C05479=1196.895,313.381,-70.607,-176.497,7.558,148.421
C05480=1196.891,313.629,-70.637,-176.494,7.561,148.421
C05481=1196.886,313.877,-70.668,-176.492,7.564,148.421
C05482=1196.882,314.126,-70.699,-176.490,7.566,148.421
C05483=1196.878,314.401,-70.733,-176.487,7.570,148.421
C05484=1196.873,314.678,-70.767,-176.484,7.573,148.421
C05485=1196.868,314.954,-70.801,-176.481,7.576,148.421
C05486=1196.864,315.230,-70.836,-176.479,7.579,148.421
C05487=1196.860,315.479,-70.867,-176.476,7.583,148.421
C05488=1196.855,315.727,-70.898,-176.474,7.585,148.421
C05489=1196.851,315.974,-70.928,-176.472,7.588,148.421
C05490=1196.847,316.223,-70.959,-176.469,7.591,148.422
C05491=1196.843,316.471,-70.990,-176.467,7.594,148.422
C05492=1196.838,316.719,-71.020,-176.465,7.596,148.422
C05493=1196.834,316.968,-71.051,-176.462,7.599,148.422
C05494=1196.830,317.215,-71.082,-176.460,7.603,148.422
C05495=1196.825,317.463,-71.112,-176.457,7.606,148.422
C05496=1196.822,317.711,-71.144,-176.455,7.608,148.422
C05497=1196.817,317.959,-71.175,-176.453,7.611,148.422
C05498=1196.812,318.207,-71.206,-176.450,7.614,148.422
C05499=1196.809,318.455,-71.236,-176.448,7.617,148.422
C05500=1196.805,318.703,-71.267,-176.445,7.620,148.422
C05501=1196.800,318.951,-71.298,-176.443,7.623,148.422
C05502=1196.796,319.199,-71.330,-176.440,7.626,148.422
C05503=1196.792,319.447,-71.360,-176.438,7.628,148.422
C05504=1196.788,319.696,-71.392,-176.436,7.631,148.422
C05505=1196.783,319.944,-71.422,-176.433,7.634,148.422
C05506=1196.779,320.191,-71.454,-176.431,7.638,148.422
C05507=1196.775,320.440,-71.484,-176.429,7.640,148.422
C05508=1196.771,320.688,-71.515,-176.426,7.643,148.422
C05509=1196.767,320.936,-71.547,-176.424,7.646,148.423
C05510=1196.763,321.184,-71.578,-176.421,7.649,148.423
C05511=1196.758,321.432,-71.609,-176.419,7.652,148.423
C05512=1196.754,321.680,-71.640,-176.417,7.655,148.423
C05513=1196.750,321.928,-71.671,-176.414,7.658,148.423
C05514=1196.746,322.176,-71.702,-176.412,7.661,148.423
C05515=1196.741,322.424,-71.734,-176.410,7.663,148.423
C05516=1196.737,322.672,-71.765,-176.407,7.667,148.423
C05517=1196.733,322.920,-71.796,-176.405,7.670,148.423
C05518=1196.729,323.168,-71.827,-176.402,7.673,148.423
C05519=1196.725,323.416,-71.859,-176.400,7.675,148.423
C05520=1196.720,323.664,-71.890,-176.398,7.678,148.423
C05521=1196.716,323.912,-71.921,-176.395,7.682,148.423
C05522=1196.712,324.160,-71.952,-176.393,7.685,148.423
C05523=1196.708,324.408,-71.983,-176.391,7.687,148.424
C05524=1196.703,324.656,-72.015,-176.388,7.690,148.424
C05525=1196.700,324.904,-72.047,-176.386,7.694,148.424
C05526=1196.695,325.152,-72.078,-176.383,7.697,148.424
C05527=1196.691,325.400,-72.109,-176.381,7.699,148.424
C05528=1196.687,325.648,-72.140,-176.379,7.702,148.424
C05529=1196.683,325.896,-72.172,-176.376,7.705,148.424
C05530=1196.678,326.144,-72.203,-176.374,7.708,148.424
C05531=1196.675,326.392,-72.235,-176.372,7.711,148.424
C05532=1196.669,326.640,-72.266,-176.370,7.714,148.424
C05533=1196.666,326.888,-72.298,-176.367,7.717,148.424
C05534=1196.662,327.136,-72.330,-176.365,7.720,148.425
C05535=1196.657,327.384,-72.360,-176.362,7.723,148.425
C05536=1196.654,327.632,-72.392,-176.360,7.726,148.425
C05537=1196.649,327.879,-72.424,-176.358,7.729,148.425
C05538=1196.645,328.128,-72.455,-176.356,7.732,148.425
C05539=1196.641,328.375,-72.486,-176.353,7.735,148.425
C05540=1196.637,328.624,-72.519,-176.351,7.738,148.425
C05541=1196.632,328.871,-72.550,-176.349,7.741,148.425
C05542=1196.628,329.120,-72.581,-176.346,7.744,148.425
C05543=1196.625,329.368,-72.613,-176.344,7.747,148.425
C05544=1196.620,329.615,-72.645,-176.342,7.750,148.425
C05545=1196.616,329.863,-72.677,-176.340,7.753,148.426
C05546=1196.611,330.111,-72.708,-176.337,7.756,148.426
C05547=1196.607,330.359,-72.740,-176.335,7.759,148.426
C05548=1196.603,330.607,-72.771,-176.333,7.761,148.426
C05549=1196.599,330.855,-72.804,-176.330,7.765,148.426
C05550=1196.595,331.103,-72.836,-176.328,7.768,148.426
C05551=1196.590,331.351,-72.866,-176.325,7.771,148.426
C05552=1196.587,331.599,-72.898,-176.324,7.774,148.426
C05553=1196.582,331.847,-72.930,-176.321,7.777,148.426
C05554=1196.578,332.095,-72.962,-176.319,7.780,148.427
C05555=1196.574,332.343,-72.994,-176.317,7.783,148.427
C05556=1196.570,332.590,-73.025,-176.314,7.786,148.427
C05557=1196.565,332.838,-73.058,-176.312,7.789,148.427
C05558=1196.562,333.086,-73.090,-176.310,7.792,148.427
C05559=1196.557,333.334,-73.121,-176.307,7.795,148.427
C05560=1196.553,333.582,-73.154,-176.305,7.799,148.427
C05561=1196.549,333.831,-73.185,-176.303,7.801,148.428
C05562=1196.545,334.078,-73.216,-176.301,7.804,148.428
C05563=1196.540,334.327,-73.249,-176.298,7.807,148.428
C05564=1196.537,334.575,-73.280,-176.296,7.811,148.428
C05565=1196.531,334.822,-73.313,-176.294,7.813,148.428
C05566=1196.528,335.070,-73.345,-176.292,7.816,148.428
C05567=1196.524,335.318,-73.377,-176.290,7.820,148.428
C05568=1196.519,335.565,-73.409,-176.287,7.823,148.428
C05569=1196.516,335.813,-73.441,-176.285,7.826,148.429
C05570=1196.512,336.061,-73.473,-176.283,7.828,148.429
C05571=1196.507,336.309,-73.505,-176.280,7.831,148.429
C05572=1196.503,336.557,-73.537,-176.278,7.835,148.429
C05573=1196.499,336.805,-73.569,-176.276,7.838,148.429
C05574=1196.495,337.053,-73.601,-176.274,7.841,148.429
C05575=1196.490,337.301,-73.633,-176.272,7.844,148.429
C05576=1196.486,337.549,-73.665,-176.269,7.847,148.430
C05577=1196.482,337.797,-73.698,-176.267,7.850,148.430
C05578=1196.478,338.045,-73.730,-176.265,7.853,148.430
C05579=1196.474,338.292,-73.761,-176.263,7.856,148.430
C05580=1196.470,338.541,-73.794,-176.260,7.859,148.430
C05581=1196.466,338.789,-73.826,-176.258,7.862,148.431
C05582=1196.462,339.036,-73.859,-176.256,7.866,148.431
C05583=1196.458,339.284,-73.890,-176.254,7.868,148.431
C05584=1196.453,339.532,-73.923,-176.252,7.871,148.431
C05585=1196.449,339.780,-73.955,-176.249,7.875,148.431
C05586=1196.445,340.028,-73.988,-176.247,7.878,148.431
C05587=1196.440,340.306,-74.023,-176.245,7.881,148.432
C05588=1196.435,340.585,-74.060,-176.243,7.885,148.432
C05589=1196.431,340.863,-74.096,-176.240,7.888,148.432
C05590=1196.426,341.142,-74.133,-176.237,7.892,148.432
C05591=1196.421,341.390,-74.165,-176.236,7.894,148.432
C05592=1196.418,341.637,-74.198,-176.233,7.898,148.432
C05593=1196.414,341.885,-74.230,-176.231,7.901,148.433
C05594=1196.410,342.133,-74.262,-176.229,7.904,148.433
C05595=1196.406,342.381,-74.295,-176.227,7.907,148.433
C05596=1196.401,342.629,-74.327,-176.225,7.910,148.433
C05597=1196.397,342.877,-74.359,-176.223,7.914,148.434
C05598=1196.393,343.125,-74.392,-176.221,7.917,148.434
C05599=1196.388,343.373,-74.424,-176.218,7.919,148.434
C05600=1196.385,343.620,-74.457,-176.216,7.922,148.434
C05601=1196.381,343.869,-74.489,-176.214,7.926,148.434
C05602=1196.376,344.116,-74.522,-176.212,7.929,148.434
C05603=1196.372,344.364,-74.554,-176.210,7.932,148.435
C05604=1196.368,344.611,-74.587,-176.208,7.935,148.435
C05605=1196.364,344.860,-74.620,-176.206,7.938,148.435
C05606=1196.360,345.107,-74.652,-176.203,7.942,148.435
C05607=1196.356,345.356,-74.685,-176.201,7.945,148.435
C05608=1196.352,345.603,-74.718,-176.199,7.947,148.436
C05609=1196.347,345.851,-74.749,-176.197,7.951,148.436
C05610=1196.343,346.098,-74.783,-176.195,7.954,148.436
C05611=1196.339,346.346,-74.816,-176.193,7.957,148.436
C05612=1196.335,346.594,-74.848,-176.191,7.960,148.436
C05613=1196.331,346.842,-74.881,-176.189,7.963,148.437
C05614=1196.327,347.090,-74.913,-176.187,7.967,148.437
C05615=1196.323,347.338,-74.946,-176.184,7.970,148.437
C05616=1196.318,347.586,-74.979,-176.183,7.972,148.437
C05617=1196.315,347.834,-75.011,-176.180,7.976,148.438
C05618=1196.311,348.081,-75.044,-176.178,7.979,148.438
C05619=1196.306,348.328,-75.077,-176.176,7.983,148.438
C05620=1196.301,348.577,-75.110,-176.175,7.985,148.438
C05621=1196.297,348.825,-75.143,-176.172,7.989,148.439
C05622=1196.294,349.072,-75.175,-176.170,7.992,148.439
C05623=1196.289,349.320,-75.208,-176.168,7.995,148.439
C05624=1196.285,349.568,-75.241,-176.166,7.999,148.439
C05625=1196.281,349.816,-75.274,-176.164,8.001,148.439
C05626=1196.277,350.064,-75.307,-176.162,8.004,148.440
C05627=1196.273,350.311,-75.340,-176.160,8.008,148.440
C05628=1196.268,350.560,-75.373,-176.158,8.011,148.440
C05629=1196.265,350.807,-75.405,-176.156,8.014,148.440
C05630=1196.261,351.055,-75.439,-176.154,8.017,148.441
C05631=1196.257,351.302,-75.472,-176.152,8.020,148.441
C05632=1196.253,351.550,-75.505,-176.150,8.024,148.441
C05633=1196.248,351.799,-75.537,-176.148,8.027,148.442
C05634=1196.244,352.046,-75.571,-176.146,8.030,148.442
C05635=1196.240,352.294,-75.604,-176.144,8.033,148.442
C05636=1196.236,352.542,-75.637,-176.142,8.037,148.442
C05637=1196.232,352.789,-75.670,-176.140,8.039,148.443
C05638=1196.227,353.037,-75.703,-176.138,8.043,148.443
C05639=1196.224,353.285,-75.736,-176.136,8.046,148.443
C05640=1196.220,353.532,-75.769,-176.134,8.049,148.443
C05641=1196.216,353.780,-75.802,-176.132,8.052,148.444
C05642=1196.212,354.028,-75.835,-176.130,8.056,148.444
C05643=1196.208,354.276,-75.868,-176.128,8.059,148.444
C05644=1196.203,354.523,-75.901,-176.126,8.062,148.444
C05645=1196.199,354.771,-75.935,-176.125,8.065,148.445
C05646=1196.195,355.019,-75.968,-176.122,8.068,148.445
C05647=1196.191,355.266,-76.001,-176.120,8.072,148.445
C05648=1196.187,355.514,-76.034,-176.118,8.075,148.446
C05649=1196.183,355.762,-76.067,-176.117,8.078,148.446
C05650=1196.179,356.010,-76.100,-176.114,8.081,148.446
C05651=1196.174,356.257,-76.134,-176.113,8.085,148.446
C05652=1196.171,356.506,-76.167,-176.110,8.088,148.447
C05653=1196.167,356.754,-76.200,-176.109,8.091,148.447
C05654=1196.163,357.001,-76.233,-176.107,8.094,148.447
C05655=1196.158,357.249,-76.267,-176.105,8.098,148.447
C05656=1196.154,357.497,-76.300,-176.103,8.101,148.448
C05657=1196.149,357.745,-76.333,-176.101,8.104,148.448
C05658=1196.146,357.992,-76.367,-176.099,8.107,148.449
C05659=1196.141,358.240,-76.400,-176.097,8.111,148.449
C05660=1196.137,358.487,-76.434,-176.095,8.114,148.449
C05661=1196.133,358.735,-76.467,-176.094,8.117,148.449
C05662=1196.130,358.984,-76.500,-176.092,8.120,148.450
C05663=1196.126,359.231,-76.534,-176.090,8.124,148.450
C05664=1196.122,359.478,-76.567,-176.088,8.127,148.450
C05665=1196.118,359.726,-76.600,-176.086,8.130,148.451
C05666=1196.113,359.974,-76.634,-176.084,8.134,148.451
C05667=1196.109,360.221,-76.668,-176.082,8.137,148.451
C05668=1196.105,360.469,-76.701,-176.081,8.140,148.452
C05669=1196.101,360.717,-76.735,-176.079,8.143,148.452
C05670=1196.097,360.965,-76.768,-176.077,8.147,148.452
C05671=1196.093,361.212,-76.802,-176.076,8.149,148.453
C05672=1196.088,361.460,-76.836,-176.074,8.153,148.453
C05673=1196.084,361.708,-76.869,-176.072,8.156,148.453
C05674=1196.080,361.955,-76.903,-176.070,8.159,148.454
C05675=1196.077,362.204,-76.936,-176.068,8.163,148.454
C05676=1196.073,362.451,-76.969,-176.067,8.166,148.454
C05677=1196.068,362.699,-77.004,-176.065,8.169,148.455
C05678=1196.064,362.946,-77.037,-176.063,8.172,148.455
C05679=1196.060,363.194,-77.070,-176.061,8.176,148.456
C05680=1196.057,363.442,-77.104,-176.060,8.179,148.456
C05681=1196.052,363.690,-77.137,-176.058,8.182,148.456
C05682=1196.048,363.937,-77.172,-176.057,8.185,148.457
C05683=1196.044,364.185,-77.205,-176.055,8.189,148.457
C05684=1196.040,364.432,-77.239,-176.053,8.192,148.457
C05685=1196.036,364.680,-77.272,-176.051,8.195,148.458
C05686=1196.032,364.928,-77.307,-176.050,8.198,148.458
C05687=1196.028,365.176,-77.340,-176.048,8.201,148.458
C05688=1196.024,365.423,-77.374,-176.047,8.205,148.459
C05689=1196.020,365.671,-77.408,-176.045,8.208,148.459
C05690=1196.016,365.918,-77.442,-176.044,8.211,148.460
C05691=1196.011,366.200,-77.480,-176.041,8.215,148.460
C05692=1196.006,366.480,-77.518,-176.040,8.218,148.460
C05693=1196.002,366.762,-77.557,-176.038,8.222,148.461
C05694=1195.998,367.042,-77.595,-176.036,8.226,148.461
C05695=1195.993,367.290,-77.629,-176.034,8.229,148.462
C05696=1195.989,367.537,-77.663,-176.033,8.232,148.462
C05697=1195.985,367.786,-77.697,-176.031,8.235,148.462
C05698=1195.981,368.033,-77.731,-176.030,8.238,148.463
C05699=1195.977,368.280,-77.764,-176.028,8.242,148.463
C05700=1195.972,368.528,-77.798,-176.027,8.245,148.464
C05701=1195.969,368.776,-77.832,-176.025,8.248,148.464
C05702=1195.965,369.023,-77.866,-176.024,8.251,148.465
C05703=1195.960,369.271,-77.900,-176.022,8.255,148.465
C05704=1195.957,369.519,-77.934,-176.021,8.258,148.465
C05705=1195.952,369.767,-77.968,-176.019,8.261,148.466
C05706=1195.948,370.014,-78.002,-176.018,8.264,148.466
C05707=1195.944,370.261,-78.036,-176.016,8.268,148.467
C05708=1195.941,370.509,-78.071,-176.015,8.271,148.467
C05709=1195.936,370.757,-78.104,-176.014,8.274,148.468
C05710=1195.932,371.004,-78.138,-176.012,8.277,148.468
C05711=1195.929,371.252,-78.172,-176.011,8.281,148.468
C05712=1195.924,371.500,-78.207,-176.009,8.284,148.469
C05713=1195.920,371.747,-78.240,-176.008,8.286,148.469
C05714=1195.916,371.995,-78.275,-176.006,8.290,148.470
C05715=1195.912,372.243,-78.309,-176.006,8.293,148.470
C05716=1195.908,372.490,-78.343,-176.004,8.297,148.471
C05717=1195.904,372.738,-78.377,-176.002,8.300,148.471
C05718=1195.899,372.986,-78.411,-176.001,8.302,148.471
C05719=1195.896,373.233,-78.445,-175.999,8.306,148.472
C05720=1195.892,373.481,-78.480,-175.999,8.309,148.472
C05721=1195.888,373.728,-78.514,-175.997,8.312,148.473
C05722=1195.884,373.976,-78.549,-175.996,8.316,148.473
C05723=1195.880,374.224,-78.582,-175.994,8.318,148.474
C05724=1195.875,374.471,-78.616,-175.994,8.322,148.474
C05725=1195.872,374.719,-78.651,-175.992,8.325,148.475
C05726=1195.867,374.967,-78.685,-175.991,8.328,148.475
C05727=1195.864,375.214,-78.719,-175.990,8.331,148.476
C05728=1195.860,375.462,-78.754,-175.989,8.334,148.476
C05729=1195.856,375.709,-78.788,-175.987,8.337,148.477
C05730=1195.852,375.957,-78.822,-175.986,8.341,148.477
C05731=1195.847,376.205,-78.857,-175.985,8.343,148.478
C05732=1195.843,376.452,-78.891,-175.983,8.347,148.478
C05733=1195.839,376.700,-78.926,-175.982,8.350,148.479
C05734=1195.835,376.948,-78.959,-175.981,8.353,148.479
C05735=1195.831,377.196,-78.994,-175.980,8.356,148.480
C05736=1195.827,377.443,-79.027,-175.979,8.359,148.480
C05737=1195.823,377.690,-79.062,-175.978,8.363,148.481
C05738=1195.819,377.938,-79.097,-175.976,8.366,148.481
C05739=1195.815,378.185,-79.131,-175.976,8.369,148.482
C05740=1195.811,378.434,-79.165,-175.974,8.371,148.482
C05741=1195.807,378.681,-79.200,-175.974,8.375,148.482
C05742=1195.803,378.927,-79.234,-175.972,8.377,148.483
C05743=1195.799,379.176,-79.269,-175.971,8.381,148.484
C05744=1195.795,379.423,-79.304,-175.970,8.384,148.484
C05745=1195.791,379.671,-79.338,-175.969,8.387,148.485
C05746=1195.787,379.918,-79.372,-175.968,8.390,148.485
C05747=1195.783,380.166,-79.407,-175.967,8.393,148.485
C05748=1195.779,380.413,-79.441,-175.966,8.396,148.486
C05749=1195.775,380.662,-79.476,-175.965,8.399,148.486
C05750=1195.770,380.909,-79.510,-175.964,8.402,148.487
C05751=1195.767,381.156,-79.544,-175.963,8.405,148.487
C05752=1195.763,381.404,-79.579,-175.962,8.408,148.488
C05753=1195.758,381.652,-79.614,-175.961,8.411,148.489
C05754=1195.755,381.899,-79.649,-175.960,8.414,148.489
C05755=1195.750,382.146,-79.683,-175.959,8.417,148.490
C05756=1195.747,382.394,-79.718,-175.959,8.420,148.490
C05757=1195.742,382.642,-79.752,-175.957,8.423,148.491
C05758=1195.739,382.890,-79.787,-175.957,8.426,148.491
C05759=1195.734,383.137,-79.821,-175.956,8.429,148.492
C05760=1195.730,383.384,-79.857,-175.955,8.432,148.492
C05761=1195.727,383.632,-79.891,-175.954,8.435,148.493
C05762=1195.723,383.880,-79.925,-175.953,8.438,148.493
C05763=1195.718,384.127,-79.960,-175.952,8.441,148.494
C05764=1195.714,384.375,-79.995,-175.951,8.444,148.494
C05765=1195.711,384.622,-80.029,-175.950,8.447,148.495
C05766=1195.707,384.870,-80.064,-175.949,8.450,148.495
C05767=1195.702,385.117,-80.099,-175.949,8.453,148.496
C05768=1195.698,385.365,-80.133,-175.947,8.456,148.496
C05769=1195.694,385.612,-80.169,-175.947,8.458,148.497
C05770=1195.691,385.860,-80.203,-175.946,8.461,148.498
C05771=1195.686,386.107,-80.237,-175.946,8.465,148.498
C05772=1195.682,386.355,-80.273,-175.945,8.468,148.499
C05773=1195.678,386.602,-80.307,-175.944,8.471,148.499
C05774=1195.674,386.850,-80.342,-175.943,8.473,148.500
C05775=1195.670,387.098,-80.376,-175.943,8.476,148.500
C05776=1195.666,387.345,-80.412,-175.942,8.479,148.501
C05777=1195.662,387.593,-80.446,-175.941,8.482,148.501
C05778=1195.658,387.841,-80.481,-175.941,8.484,148.502
C05779=1195.654,388.088,-80.516,-175.940,8.487,148.503
C05780=1195.650,388.335,-80.550,-175.939,8.491,148.503
C05781=1195.646,388.583,-80.585,-175.938,8.494,148.504
C05782=1195.642,388.830,-80.620,-175.938,8.496,148.504
C05783=1195.638,389.078,-80.655,-175.937,8.499,148.505
C05784=1195.634,389.325,-80.690,-175.936,8.502,148.505
C05785=1195.630,389.573,-80.725,-175.936,8.504,148.506
C05786=1195.626,389.820,-80.759,-175.935,8.507,148.506
C05787=1195.622,390.068,-80.795,-175.935,8.509,148.507
C05788=1195.618,390.316,-80.829,-175.934,8.513,148.507
C05789=1195.614,390.563,-80.865,-175.933,8.516,148.508
C05790=1195.610,390.811,-80.899,-175.933,8.518,148.509
C05791=1195.606,391.058,-80.934,-175.932,8.521,148.509
C05792=1195.602,391.306,-80.969,-175.932,8.523,148.510
C05793=1195.597,391.553,-81.004,-175.931,8.526,148.510
C05794=1195.594,391.800,-81.039,-175.931,8.529,148.511
C05795=1195.589,392.084,-81.078,-175.930,8.532,148.511
C05796=1195.585,392.367,-81.119,-175.930,8.535,148.512
C05797=1195.580,392.650,-81.158,-175.929,8.538,148.513
C05798=1195.576,392.933,-81.199,-175.928,8.541,148.513
C05799=1195.571,393.181,-81.234,-175.928,8.544,148.514
C05800=1195.568,393.428,-81.269,-175.927,8.547,148.514
C05801=1195.564,393.676,-81.303,-175.927,8.549,148.515
C05802=1195.560,393.923,-81.339,-175.926,8.552,148.516
C05803=1195.556,394.171,-81.373,-175.926,8.554,148.516
C05804=1195.552,394.418,-81.409,-175.925,8.557,148.517
C05805=1195.548,394.666,-81.443,-175.925,8.560,148.517
C05806=1195.544,394.913,-81.479,-175.924,8.563,148.518
C05807=1195.540,395.161,-81.513,-175.924,8.565,148.518
C05808=1195.536,395.408,-81.549,-175.924,8.567,148.519
C05809=1195.531,395.656,-81.583,-175.923,8.570,148.519
C05810=1195.528,395.903,-81.619,-175.923,8.573,148.520
C05811=1195.524,396.151,-81.655,-175.923,8.575,148.521
C05812=1195.519,396.398,-81.689,-175.922,8.578,148.521
C05813=1195.516,396.646,-81.725,-175.922,8.581,148.522
C05814=1195.512,396.894,-81.759,-175.922,8.583,148.522
C05815=1195.508,397.141,-81.795,-175.921,8.586,148.523
C05816=1195.504,397.389,-81.829,-175.921,8.588,148.523
C05817=1195.499,397.636,-81.865,-175.920,8.591,148.524
C05818=1195.496,397.883,-81.900,-175.920,8.594,148.525
C05819=1195.492,398.131,-81.935,-175.919,8.596,148.525
C05820=1195.487,398.378,-81.970,-175.919,8.598,148.526
C05821=1195.483,398.626,-82.005,-175.919,8.600,148.526
C05822=1195.480,398.874,-82.041,-175.918,8.604,148.527
C05823=1195.476,399.120,-82.076,-175.918,8.606,148.527
C05824=1195.472,399.369,-82.111,-175.918,8.608,148.528
C05825=1195.468,399.616,-82.146,-175.917,8.610,148.528
C05826=1195.464,399.863,-82.181,-175.917,8.613,148.529
C05827=1195.460,400.111,-82.216,-175.916,8.616,148.529
C05828=1195.455,400.358,-82.251,-175.916,8.618,148.530
C05829=1195.452,400.605,-82.287,-175.916,8.621,148.531
C05830=1195.448,400.853,-82.322,-175.916,8.623,148.531
C05831=1195.443,401.100,-82.357,-175.915,8.626,148.532
C05832=1195.440,401.348,-82.392,-175.915,8.628,148.532
C05833=1195.436,401.596,-82.427,-175.915,8.630,148.533
C05834=1195.432,401.843,-82.462,-175.915,8.633,148.533
C05835=1195.428,402.090,-82.498,-175.914,8.635,148.534
C05836=1195.424,402.338,-82.533,-175.914,8.637,148.535
C05837=1195.420,402.585,-82.568,-175.914,8.640,148.535
C05838=1195.416,402.832,-82.604,-175.913,8.643,148.536
C05839=1195.412,403.081,-82.638,-175.913,8.645,148.536
C05840=1195.408,403.327,-82.674,-175.913,8.647,148.537
C05841=1195.404,403.575,-82.709,-175.912,8.649,148.537
C05842=1195.400,403.822,-82.745,-175.912,8.652,148.538
C05843=1195.396,404.071,-82.780,-175.912,8.654,148.538
C05844=1195.392,404.318,-82.815,-175.912,8.656,148.539
C05845=1195.388,404.565,-82.851,-175.911,8.659,148.539
C05846=1195.384,404.813,-82.886,-175.911,8.661,148.540
C05847=1195.380,405.060,-82.921,-175.911,8.663,148.540
C05848=1195.376,405.308,-82.956,-175.911,8.665,148.541
C05849=1195.372,405.555,-82.992,-175.911,8.668,148.541
C05850=1195.368,405.802,-83.027,-175.911,8.670,148.542
C05851=1195.364,406.050,-83.062,-175.911,8.672,148.543
C05852=1195.360,406.297,-83.097,-175.910,8.675,148.543
C05853=1195.356,406.544,-83.133,-175.910,8.677,148.544
C05854=1195.352,406.792,-83.168,-175.910,8.679,148.544
C05855=1195.348,407.040,-83.204,-175.910,8.681,148.545
C05856=1195.344,407.288,-83.239,-175.909,8.684,148.545
C05857=1195.340,407.535,-83.274,-175.909,8.686,148.546
C05858=1195.336,407.782,-83.310,-175.909,8.688,148.546
C05859=1195.333,408.030,-83.345,-175.909,8.691,148.547
C05860=1195.328,408.277,-83.380,-175.908,8.693,148.547
C05861=1195.324,408.524,-83.415,-175.908,8.695,148.548
C05862=1195.321,408.772,-83.451,-175.908,8.697,148.548
C05863=1195.316,409.020,-83.487,-175.908,8.700,148.549
C05864=1195.312,409.267,-83.522,-175.907,8.702,148.550
C05865=1195.308,409.514,-83.558,-175.907,8.704,148.550
C05866=1195.304,409.762,-83.593,-175.907,8.706,148.551
C05867=1195.301,410.010,-83.628,-175.907,8.708,148.551
C05868=1195.296,410.256,-83.663,-175.907,8.710,148.552
C05869=1195.293,410.504,-83.699,-175.907,8.712,148.552
C05870=1195.289,410.751,-83.735,-175.907,8.715,148.553
C05871=1195.284,410.999,-83.770,-175.906,8.717,148.553
C05872=1195.280,411.246,-83.806,-175.906,8.719,148.554
C05873=1195.277,411.494,-83.841,-175.905,8.721,148.554
C05874=1195.273,411.742,-83.876,-175.905,8.723,148.555
C05875=1195.269,411.988,-83.911,-175.905,8.725,148.555
C05876=1195.265,412.236,-83.947,-175.905,8.727,148.556
C05877=1195.260,412.484,-83.983,-175.905,8.729,148.556
C05878=1195.257,412.731,-84.019,-175.905,8.732,148.557
C05879=1195.253,412.978,-84.054,-175.904,8.734,148.557
C05880=1195.249,413.226,-84.089,-175.904,8.736,148.558
C05881=1195.245,413.473,-84.125,-175.905,8.738,148.558
C05882=1195.241,413.721,-84.161,-175.904,8.740,148.559
C05883=1195.237,413.968,-84.196,-175.904,8.742,148.559
C05884=1195.233,414.216,-84.231,-175.904,8.744,148.560
C05885=1195.229,414.463,-84.267,-175.904,8.747,148.560
C05886=1195.225,414.711,-84.302,-175.904,8.748,148.561
C05887=1195.221,414.958,-84.337,-175.904,8.750,148.561
C05888=1195.217,415.205,-84.374,-175.903,8.752,148.562
C05889=1195.213,415.453,-84.409,-175.903,8.755,148.562
C05890=1195.209,415.700,-84.445,-175.902,8.757,148.563
C05891=1195.203,416.053,-84.495,-175.903,8.759,148.563
C05892=1195.199,416.405,-84.546,-175.902,8.763,148.564
C05893=1195.199,416.758,-84.597,-175.902,8.765,148.565
C05894=1195.202,417.110,-84.645,-175.902,8.767,148.565
C05895=1194.780,417.110,-84.686,-175.905,8.778,148.569
C05896=1194.777,416.756,-84.635,-175.905,8.776,148.568
C05897=1194.778,416.400,-84.584,-175.905,8.773,148.568
C05898=1194.782,416.045,-84.534,-175.906,8.770,148.567
C05899=1194.787,415.689,-84.482,-175.906,8.768,148.566
C05900=1194.791,415.443,-84.447,-175.906,8.765,148.566
C05901=1194.796,415.194,-84.412,-175.906,8.763,148.565
C05902=1194.800,414.947,-84.376,-175.906,8.761,148.565
C05903=1194.803,414.699,-84.341,-175.907,8.759,148.564
C05904=1194.807,414.452,-84.305,-175.907,8.757,148.564
C05905=1194.811,414.205,-84.270,-175.907,8.755,148.563
C05906=1194.816,413.957,-84.234,-175.907,8.753,148.563
C05907=1194.819,413.710,-84.198,-175.907,8.751,148.562
C05908=1194.823,413.462,-84.163,-175.908,8.748,148.562
C05909=1194.827,413.215,-84.127,-175.907,8.747,148.561
C05910=1194.831,412.968,-84.092,-175.908,8.745,148.561
C05911=1194.835,412.720,-84.056,-175.908,8.742,148.560
C05912=1194.839,412.472,-84.020,-175.908,8.740,148.560
C05913=1194.843,412.226,-83.985,-175.908,8.738,148.559
C05914=1194.847,411.978,-83.949,-175.909,8.735,148.559
C05915=1194.851,411.730,-83.915,-175.908,8.734,148.558
C05916=1194.855,411.483,-83.879,-175.908,8.732,148.558
C05917=1194.860,411.235,-83.843,-175.909,8.730,148.557
C05918=1194.863,410.988,-83.808,-175.909,8.727,148.557
C05919=1194.867,410.740,-83.772,-175.909,8.725,148.556
C05920=1194.871,410.494,-83.737,-175.909,8.723,148.556
C05921=1194.875,410.246,-83.701,-175.910,8.720,148.555
C05922=1194.878,409.999,-83.666,-175.909,8.719,148.555
C05923=1194.883,409.750,-83.631,-175.910,8.717,148.554
C05924=1194.887,409.503,-83.595,-175.910,8.714,148.554
C05925=1194.891,409.256,-83.560,-175.910,8.712,148.553
C05926=1194.895,409.008,-83.524,-175.910,8.710,148.552
C05927=1194.898,408.761,-83.489,-175.911,8.708,148.552
C05928=1194.903,408.514,-83.453,-175.911,8.705,148.551
C05929=1194.907,408.266,-83.419,-175.911,8.703,148.551
C05930=1194.911,408.018,-83.383,-175.911,8.701,148.550
C05931=1194.915,407.771,-83.347,-175.912,8.699,148.550
C05932=1194.919,407.524,-83.312,-175.912,8.696,148.549
C05933=1194.923,407.276,-83.276,-175.912,8.694,148.549
C05934=1194.926,407.029,-83.241,-175.912,8.692,148.548
C05935=1194.931,406.781,-83.206,-175.913,8.690,148.548
C05936=1194.935,406.534,-83.171,-175.913,8.687,148.547
C05937=1194.938,406.286,-83.135,-175.913,8.685,148.547
C05938=1194.942,406.040,-83.100,-175.913,8.683,148.546
C05939=1194.947,405.792,-83.064,-175.913,8.681,148.546
C05940=1194.951,405.544,-83.029,-175.914,8.678,148.545
C05941=1194.955,405.296,-82.993,-175.914,8.676,148.545
C05942=1194.959,405.049,-82.958,-175.914,8.674,148.544
C05943=1194.962,404.802,-82.923,-175.914,8.671,148.544
C05944=1194.966,404.554,-82.888,-175.915,8.669,148.543
C05945=1194.971,404.307,-82.853,-175.915,8.667,148.542
C05946=1194.974,404.059,-82.817,-175.915,8.665,148.542
C05947=1194.978,403.812,-82.782,-175.915,8.662,148.541
C05948=1194.983,403.565,-82.747,-175.916,8.660,148.541
C05949=1194.986,403.317,-82.712,-175.916,8.658,148.540
C05950=1194.990,403.070,-82.676,-175.916,8.656,148.540
C05951=1194.994,402.823,-82.641,-175.916,8.653,148.539
C05952=1194.999,402.574,-82.605,-175.916,8.651,148.539
C05953=1195.003,402.327,-82.570,-175.916,8.648,148.538
C05954=1195.007,402.080,-82.535,-175.917,8.646,148.538
C05955=1195.011,401.832,-82.500,-175.917,8.643,148.537
C05956=1195.014,401.584,-82.464,-175.918,8.641,148.536
C05957=1195.019,401.338,-82.429,-175.918,8.639,148.536
C05958=1195.023,401.089,-82.394,-175.918,8.636,148.535
C05959=1195.026,400.842,-82.359,-175.918,8.634,148.535
C05960=1195.031,400.595,-82.324,-175.919,8.632,148.534
C05961=1195.035,400.347,-82.289,-175.919,8.629,148.534
C05962=1195.038,400.100,-82.253,-175.920,8.626,148.533
C05963=1195.042,399.853,-82.218,-175.920,8.624,148.533
C05964=1195.046,399.605,-82.183,-175.920,8.622,148.532
C05965=1195.050,399.357,-82.148,-175.920,8.620,148.532
C05966=1195.054,399.110,-82.112,-175.921,8.616,148.531
C05967=1195.058,398.862,-82.078,-175.921,8.614,148.530
C05968=1195.062,398.615,-82.042,-175.921,8.612,148.530
C05969=1195.066,398.368,-82.007,-175.921,8.609,148.529
C05970=1195.070,398.120,-81.972,-175.922,8.606,148.529
C05971=1195.074,397.872,-81.937,-175.922,8.604,148.528
C05972=1195.078,397.625,-81.902,-175.923,8.602,148.528
C05973=1195.082,397.377,-81.866,-175.923,8.599,148.527
C05974=1195.086,397.130,-81.831,-175.924,8.596,148.526
C05975=1195.090,396.882,-81.796,-175.924,8.594,148.526
C05976=1195.094,396.635,-81.761,-175.924,8.592,148.525
C05977=1195.099,396.388,-81.726,-175.925,8.589,148.525
C05978=1195.102,396.140,-81.691,-175.925,8.586,148.524
C05979=1195.106,395.893,-81.655,-175.925,8.584,148.524
C05980=1195.110,395.645,-81.621,-175.926,8.581,148.523
C05981=1195.114,395.398,-81.585,-175.926,8.579,148.523
C05982=1195.119,395.150,-81.551,-175.927,8.575,148.522
C05983=1195.122,394.903,-81.515,-175.927,8.573,148.521
C05984=1195.126,394.655,-81.481,-175.927,8.571,148.521
C05985=1195.131,394.408,-81.445,-175.928,8.568,148.520
C05986=1195.135,394.160,-81.410,-175.928,8.566,148.520
C05987=1195.138,393.912,-81.375,-175.929,8.562,148.519
C05988=1195.143,393.665,-81.340,-175.929,8.560,148.519
C05989=1195.146,393.418,-81.306,-175.930,8.557,148.518
C05990=1195.150,393.170,-81.271,-175.930,8.555,148.517
C05991=1195.154,392.923,-81.236,-175.931,8.552,148.517
C05992=1195.159,392.639,-81.196,-175.931,8.549,148.516
C05993=1195.163,392.356,-81.156,-175.932,8.546,148.516
C05994=1195.168,392.073,-81.116,-175.932,8.543,148.515
C05995=1195.173,391.790,-81.075,-175.933,8.540,148.514
C05996=1195.176,391.542,-81.041,-175.934,8.537,148.514
C05997=1195.180,391.295,-81.006,-175.934,8.534,148.513
C05998=1195.184,391.047,-80.971,-175.935,8.531,148.513
C05999=1195.188,390.800,-80.936,-175.935,8.529,148.512
C06000=1195.192,390.552,-80.901,-175.936,8.526,148.512
C06001=1195.197,390.305,-80.866,-175.936,8.524,148.511
C06002=1195.201,390.057,-80.831,-175.937,8.521,148.510
C06003=1195.205,389.809,-80.796,-175.938,8.518,148.510
C06004=1195.208,389.562,-80.761,-175.938,8.515,148.509
C06005=1195.212,389.314,-80.727,-175.939,8.512,148.509
C06006=1195.216,389.068,-80.691,-175.940,8.509,148.508
C06007=1195.220,388.819,-80.657,-175.940,8.507,148.508
C06008=1195.225,388.572,-80.622,-175.941,8.504,148.507
C06009=1195.229,388.324,-80.587,-175.942,8.501,148.506
C06010=1195.233,388.077,-80.552,-175.942,8.499,148.506
C06011=1195.236,387.829,-80.518,-175.943,8.496,148.505
C06012=1195.240,387.582,-80.482,-175.944,8.492,148.505
C06013=1195.245,387.334,-80.448,-175.945,8.489,148.504
C06014=1195.249,387.086,-80.413,-175.945,8.487,148.504
C06015=1195.253,386.839,-80.378,-175.946,8.484,148.503
C06016=1195.256,386.592,-80.344,-175.946,8.481,148.503
C06017=1195.261,386.344,-80.309,-175.947,8.478,148.502
C06018=1195.264,386.097,-80.274,-175.948,8.475,148.502
C06019=1195.269,385.849,-80.239,-175.949,8.473,148.501
C06020=1195.273,385.601,-80.204,-175.949,8.470,148.501
C06021=1195.276,385.355,-80.170,-175.950,8.467,148.500
C06022=1195.280,385.107,-80.135,-175.951,8.463,148.499
C06023=1195.285,384.859,-80.100,-175.952,8.460,148.499
C06024=1195.289,384.611,-80.066,-175.953,8.458,148.498
C06025=1195.293,384.364,-80.030,-175.954,8.454,148.498
C06026=1195.296,384.116,-79.996,-175.954,8.452,148.497
C06027=1195.301,383.869,-79.962,-175.955,8.449,148.497
C06028=1195.305,383.621,-79.927,-175.956,8.446,148.496
C06029=1195.309,383.373,-79.892,-175.957,8.443,148.496
C06030=1195.312,383.126,-79.857,-175.958,8.440,148.495
C06031=1195.317,382.879,-79.823,-175.958,8.437,148.494
C06032=1195.321,382.631,-79.788,-175.960,8.434,148.494
C06033=1195.326,382.383,-79.754,-175.960,8.431,148.494
C06034=1195.329,382.135,-79.719,-175.961,8.428,148.493
C06035=1195.333,381.889,-79.684,-175.962,8.425,148.493
C06036=1195.337,381.641,-79.649,-175.963,8.422,148.492
C06037=1195.341,381.393,-79.616,-175.964,8.419,148.491
C06038=1195.345,381.145,-79.581,-175.965,8.416,148.491
C06039=1195.349,380.898,-79.546,-175.966,8.413,148.490
C06040=1195.353,380.650,-79.512,-175.967,8.410,148.490
C06041=1195.357,380.403,-79.478,-175.968,8.407,148.489
C06042=1195.362,380.155,-79.443,-175.969,8.403,148.489
C06043=1195.365,379.908,-79.408,-175.971,8.400,148.488
C06044=1195.369,379.661,-79.374,-175.971,8.397,148.488
C06045=1195.373,379.413,-79.339,-175.973,8.394,148.487
C06046=1195.378,379.165,-79.304,-175.973,8.391,148.487
C06047=1195.381,378.917,-79.270,-175.974,8.388,148.486
C06048=1195.386,378.670,-79.236,-175.975,8.385,148.486
C06049=1195.389,378.422,-79.201,-175.976,8.382,148.485
C06050=1195.393,378.175,-79.167,-175.978,8.379,148.485
C06051=1195.398,377.927,-79.132,-175.979,8.376,148.484
C06052=1195.401,377.679,-79.098,-175.980,8.373,148.484
C06053=1195.406,377.432,-79.064,-175.981,8.370,148.483
C06054=1195.410,377.184,-79.029,-175.982,8.367,148.483
C06055=1195.414,376.937,-78.995,-175.984,8.363,148.482
C06056=1195.418,376.689,-78.961,-175.985,8.360,148.482
C06057=1195.421,376.442,-78.926,-175.986,8.357,148.481
C06058=1195.426,376.194,-78.892,-175.987,8.354,148.481
C06059=1195.430,375.946,-78.857,-175.988,8.351,148.480
C06060=1195.434,375.699,-78.823,-175.990,8.348,148.480
C06061=1195.438,375.451,-78.789,-175.990,8.345,148.479
C06062=1195.441,375.204,-78.755,-175.992,8.341,148.479
C06063=1195.446,374.956,-78.721,-175.993,8.338,148.479
C06064=1195.450,374.708,-78.687,-175.994,8.335,148.478
C06065=1195.454,374.460,-78.652,-175.996,8.332,148.478
C06066=1195.458,374.213,-78.618,-175.997,8.329,148.477
C06067=1195.462,373.965,-78.583,-175.998,8.326,148.477
C06068=1195.466,373.718,-78.549,-175.999,8.323,148.476
C06069=1195.470,373.471,-78.515,-176.001,8.319,148.476
C06070=1195.474,373.223,-78.481,-176.002,8.316,148.475
C06071=1195.478,372.975,-78.447,-176.003,8.313,148.475
C06072=1195.482,372.727,-78.413,-176.005,8.310,148.474
C06073=1195.486,372.480,-78.378,-176.006,8.307,148.474
C06074=1195.490,372.232,-78.344,-176.008,8.303,148.474
C06075=1195.494,371.984,-78.310,-176.009,8.300,148.473
C06076=1195.498,371.737,-78.276,-176.010,8.297,148.473
C06077=1195.503,371.489,-78.242,-176.012,8.294,148.472
C06078=1195.506,371.241,-78.208,-176.013,8.291,148.472
C06079=1195.511,370.994,-78.173,-176.015,8.287,148.471
C06080=1195.515,370.746,-78.140,-176.016,8.285,148.471
C06081=1195.519,370.498,-78.105,-176.018,8.281,148.471
C06082=1195.523,370.251,-78.071,-176.019,8.278,148.470
C06083=1195.527,370.004,-78.037,-176.021,8.274,148.470
C06084=1195.531,369.756,-78.004,-176.022,8.271,148.469
C06085=1195.534,369.508,-77.970,-176.023,8.269,148.469
C06086=1195.539,369.261,-77.935,-176.025,8.265,148.468
C06087=1195.543,369.013,-77.902,-176.026,8.262,148.468
C06088=1195.547,368.765,-77.867,-176.028,8.258,148.467
C06089=1195.551,368.518,-77.833,-176.029,8.256,148.467
C06090=1195.555,368.270,-77.800,-176.031,8.252,148.467
C06091=1195.560,368.023,-77.766,-176.032,8.249,148.466
C06092=1195.563,367.775,-77.731,-176.034,8.246,148.466
C06093=1195.568,367.527,-77.698,-176.035,8.242,148.465
C06094=1195.572,367.280,-77.664,-176.037,8.239,148.465
C06095=1195.575,367.031,-77.630,-176.039,8.236,148.465
C06096=1195.580,366.750,-77.592,-176.041,8.232,148.464
C06097=1195.585,366.470,-77.553,-176.042,8.229,148.464
C06098=1195.589,366.189,-77.515,-176.044,8.225,148.463
C06099=1195.594,365.907,-77.477,-176.046,8.221,148.463
C06100=1195.598,365.660,-77.443,-176.047,8.218,148.463
C06101=1195.603,365.412,-77.409,-176.049,8.215,148.462
C06102=1195.606,365.165,-77.375,-176.051,8.211,148.462
C06103=1195.610,364.917,-77.342,-176.052,8.208,148.461
C06104=1195.614,364.670,-77.308,-176.054,8.205,148.461
C06105=1195.619,364.421,-77.274,-176.055,8.202,148.461
C06106=1195.622,364.174,-77.240,-176.057,8.199,148.460
C06107=1195.627,363.927,-77.207,-176.059,8.195,148.460
C06108=1195.630,363.679,-77.173,-176.060,8.192,148.459
C06109=1195.635,363.431,-77.139,-176.062,8.189,148.459
C06110=1195.639,363.184,-77.105,-176.064,8.185,148.459
C06111=1195.643,362.936,-77.072,-176.065,8.182,148.458
C06112=1195.646,362.688,-77.038,-176.067,8.179,148.458
C06113=1195.651,362.440,-77.004,-176.070,8.175,148.458
C06114=1195.655,362.192,-76.971,-176.071,8.173,148.457
C06115=1195.659,361.945,-76.937,-176.073,8.169,148.457
C06116=1195.663,361.698,-76.904,-176.075,8.166,148.457
C06117=1195.667,361.450,-76.871,-176.076,8.163,148.456
C06118=1195.671,361.202,-76.836,-176.078,8.160,148.456
C06119=1195.675,360.954,-76.803,-176.080,8.156,148.456
C06120=1195.679,360.706,-76.769,-176.081,8.153,148.455
C06121=1195.683,360.459,-76.736,-176.083,8.150,148.455
C06122=1195.687,360.211,-76.702,-176.085,8.146,148.455
C06123=1195.691,359.964,-76.669,-176.087,8.144,148.454
C06124=1195.696,359.715,-76.635,-176.089,8.140,148.454
C06125=1195.700,359.467,-76.602,-176.091,8.137,148.454
C06126=1195.704,359.220,-76.568,-176.093,8.133,148.453
C06127=1195.708,358.972,-76.535,-176.094,8.131,148.453
C06128=1195.712,358.725,-76.502,-176.096,8.127,148.453
C06129=1195.716,358.477,-76.469,-176.098,8.124,148.452
C06130=1195.720,358.229,-76.436,-176.100,8.121,148.452
C06131=1195.724,357.982,-76.402,-176.102,8.117,148.452
C06132=1195.728,357.734,-76.368,-176.104,8.114,148.451
C06133=1195.732,357.486,-76.335,-176.106,8.110,148.451
C06134=1195.737,357.238,-76.301,-176.107,8.108,148.451
C06135=1195.741,356.990,-76.268,-176.109,8.104,148.451
C06136=1195.745,356.742,-76.235,-176.112,8.101,148.450
C06137=1195.749,356.495,-76.202,-176.113,8.097,148.450
C06138=1195.753,356.248,-76.168,-176.115,8.095,148.450
C06139=1195.757,356.000,-76.135,-176.117,8.091,148.449
C06140=1195.761,355.752,-76.102,-176.119,8.088,148.449
C06141=1195.765,355.504,-76.068,-176.121,8.085,148.449
C06142=1195.769,355.257,-76.035,-176.123,8.081,148.448
C06143=1195.773,355.009,-76.002,-176.125,8.078,148.448
C06144=1195.777,354.760,-75.969,-176.127,8.075,148.448
C06145=1195.781,354.513,-75.935,-176.129,8.071,148.448
C06146=1195.785,354.265,-75.902,-176.131,8.068,148.447
C06147=1195.789,354.017,-75.869,-176.133,8.066,148.447
C06148=1195.794,353.770,-75.836,-176.135,8.062,148.447
C06149=1195.798,353.522,-75.803,-176.137,8.059,148.447
C06150=1195.802,353.274,-75.770,-176.139,8.055,148.446
C06151=1195.806,353.026,-75.737,-176.141,8.053,148.446
C06152=1195.810,352.779,-75.703,-176.142,8.049,148.446
C06153=1195.814,352.531,-75.671,-176.145,8.046,148.445
C06154=1195.818,352.283,-75.638,-176.147,8.043,148.445
C06155=1195.822,352.035,-75.605,-176.149,8.040,148.445
C06156=1195.826,351.787,-75.572,-176.151,8.037,148.445
C06157=1195.830,351.540,-75.539,-176.153,8.033,148.444
C06158=1195.835,351.292,-75.506,-176.155,8.030,148.444
C06159=1195.839,351.044,-75.473,-176.156,8.027,148.444
C06160=1195.843,350.796,-75.440,-176.159,8.024,148.444
C06161=1195.847,350.548,-75.407,-176.161,8.021,148.444
C06162=1195.851,350.300,-75.374,-176.163,8.017,148.443
C06163=1195.855,350.053,-75.341,-176.165,8.014,148.443
C06164=1195.859,349.805,-75.308,-176.167,8.011,148.443
C06165=1195.863,349.557,-75.276,-176.169,8.008,148.443
C06166=1195.867,349.309,-75.242,-176.171,8.004,148.442
C06167=1195.872,349.062,-75.210,-176.173,8.001,148.442
C06168=1195.876,348.814,-75.177,-176.175,7.999,148.442
C06169=1195.880,348.566,-75.145,-176.177,7.995,148.442
C06170=1195.884,348.319,-75.112,-176.179,7.992,148.441
C06171=1195.888,348.071,-75.078,-176.181,7.988,148.441
C06172=1195.893,347.823,-75.046,-176.183,7.986,148.441
C06173=1195.897,347.575,-75.013,-176.185,7.982,148.441
C06174=1195.900,347.327,-74.980,-176.187,7.979,148.440
C06175=1195.905,347.079,-74.948,-176.190,7.976,148.440
C06176=1195.909,346.831,-74.915,-176.192,7.973,148.440
C06177=1195.913,346.584,-74.881,-176.194,7.970,148.440
C06178=1195.917,346.336,-74.850,-176.196,7.967,148.440
C06179=1195.921,346.089,-74.817,-176.198,7.963,148.439
C06180=1195.926,345.840,-74.784,-176.200,7.960,148.439
C06181=1195.930,345.593,-74.751,-176.202,7.958,148.439
C06182=1195.933,345.345,-74.719,-176.204,7.954,148.439
C06183=1195.938,345.097,-74.686,-176.206,7.951,148.438
C06184=1195.942,344.849,-74.653,-176.209,7.948,148.438
C06185=1195.946,344.601,-74.621,-176.210,7.945,148.438
C06186=1195.950,344.353,-74.588,-176.212,7.942,148.438
C06187=1195.955,344.106,-74.556,-176.215,7.938,148.438
C06188=1195.959,343.858,-74.523,-176.217,7.935,148.437
C06189=1195.963,343.610,-74.491,-176.219,7.932,148.437
C06190=1195.967,343.362,-74.458,-176.221,7.929,148.437
C06191=1195.971,343.114,-74.426,-176.223,7.926,148.437
C06192=1195.975,342.866,-74.394,-176.226,7.923,148.437
C06193=1195.980,342.619,-74.361,-176.228,7.920,148.437
C06194=1195.984,342.371,-74.329,-176.230,7.917,148.436
C06195=1195.988,342.123,-74.296,-176.232,7.914,148.436
C06196=1195.992,341.875,-74.263,-176.234,7.910,148.436
C06197=1195.996,341.627,-74.232,-176.236,7.907,148.436
C06198=1196.001,341.379,-74.199,-176.239,7.904,148.436
C06199=1196.004,341.131,-74.167,-176.240,7.901,148.435
C06200=1196.009,340.853,-74.130,-176.244,7.897,148.435
C06201=1196.013,340.574,-74.094,-176.246,7.894,148.435
C06202=1196.018,340.295,-74.058,-176.248,7.891,148.435
C06203=1196.023,340.017,-74.022,-176.250,7.887,148.435
C06204=1196.027,339.770,-73.989,-176.252,7.884,148.434
C06205=1196.032,339.521,-73.956,-176.255,7.881,148.434
C06206=1196.035,339.273,-73.924,-176.257,7.878,148.434
C06207=1196.040,339.026,-73.892,-176.259,7.875,148.434
C06208=1196.044,338.778,-73.860,-176.261,7.872,148.434
C06209=1196.048,338.530,-73.827,-176.264,7.868,148.434
C06210=1196.052,338.282,-73.795,-176.266,7.865,148.433
C06211=1196.057,338.034,-73.763,-176.268,7.863,148.433
C06212=1196.061,337.786,-73.731,-176.270,7.860,148.433
C06213=1196.064,337.539,-73.699,-176.272,7.856,148.433
C06214=1196.068,337.290,-73.666,-176.275,7.853,148.433
C06215=1196.073,337.043,-73.635,-176.277,7.850,148.433
C06216=1196.077,336.795,-73.602,-176.279,7.847,148.433
C06217=1196.081,336.547,-73.571,-176.281,7.844,148.432
C06218=1196.086,336.299,-73.539,-176.283,7.841,148.432
C06219=1196.090,336.051,-73.507,-176.286,7.838,148.432
C06220=1196.093,335.803,-73.475,-176.288,7.835,148.432
C06221=1196.098,335.554,-73.442,-176.290,7.832,148.432
C06222=1196.102,335.308,-73.410,-176.293,7.829,148.432
C06223=1196.106,335.059,-73.378,-176.295,7.826,148.432
C06224=1196.110,334.811,-73.346,-176.297,7.822,148.431
C06225=1196.114,334.564,-73.314,-176.299,7.820,148.431
C06226=1196.119,334.316,-73.282,-176.302,7.817,148.431
C06227=1196.122,334.068,-73.250,-176.304,7.813,148.431
C06228=1196.127,333.820,-73.219,-176.306,7.810,148.431
C06229=1196.131,333.572,-73.186,-176.308,7.808,148.431
C06230=1196.135,333.324,-73.154,-176.310,7.805,148.431
C06231=1196.139,333.077,-73.123,-176.313,7.802,148.431
C06232=1196.144,332.828,-73.091,-176.315,7.798,148.430
C06233=1196.148,332.580,-73.059,-176.317,7.796,148.430
C06234=1196.152,332.332,-73.028,-176.320,7.793,148.430
C06235=1196.156,332.084,-72.995,-176.322,7.789,148.430
C06236=1196.160,331.836,-72.964,-176.324,7.786,148.430
C06237=1196.164,331.589,-72.932,-176.327,7.783,148.430
C06238=1196.169,331.340,-72.900,-176.329,7.780,148.430
C06239=1196.173,331.093,-72.868,-176.331,7.777,148.430
C06240=1196.177,330.845,-72.836,-176.333,7.774,148.429
C06241=1196.181,330.596,-72.805,-176.336,7.771,148.429
C06242=1196.186,330.348,-72.773,-176.338,7.769,148.429
C06243=1196.190,330.100,-72.741,-176.340,7.765,148.429
C06244=1196.194,329.853,-72.710,-176.343,7.762,148.429
C06245=1196.198,329.605,-72.678,-176.345,7.759,148.429
C06246=1196.202,329.356,-72.647,-176.348,7.756,148.429
C06247=1196.207,329.109,-72.615,-176.349,7.753,148.429
C06248=1196.210,328.861,-72.583,-176.352,7.750,148.428
C06249=1196.215,328.613,-72.551,-176.354,7.747,148.428
C06250=1196.219,328.365,-72.520,-176.356,7.744,148.428
C06251=1196.223,328.117,-72.489,-176.359,7.742,148.428
C06252=1196.228,327.869,-72.456,-176.361,7.738,148.428
C06253=1196.232,327.621,-72.426,-176.364,7.735,148.428
C06254=1196.236,327.373,-72.394,-176.366,7.732,148.428
C06255=1196.240,327.125,-72.362,-176.368,7.730,148.428
C06256=1196.244,326.877,-72.331,-176.370,7.726,148.428
C06257=1196.248,326.629,-72.299,-176.373,7.723,148.428
C06258=1196.252,326.381,-72.269,-176.375,7.720,148.427
C06259=1196.256,326.133,-72.237,-176.377,7.718,148.427
C06260=1196.261,325.885,-72.205,-176.379,7.714,148.427
C06261=1196.265,325.637,-72.174,-176.382,7.711,148.427
C06262=1196.270,325.389,-72.142,-176.384,7.708,148.427
C06263=1196.274,325.141,-72.111,-176.387,7.705,148.427
C06264=1196.278,324.893,-72.079,-176.389,7.703,148.427
C06265=1196.282,324.645,-72.048,-176.391,7.700,148.427
C06266=1196.286,324.397,-72.017,-176.394,7.697,148.427
C06267=1196.290,324.149,-71.986,-176.396,7.693,148.427
C06268=1196.294,323.901,-71.954,-176.398,7.691,148.427
C06269=1196.299,323.653,-71.923,-176.401,7.688,148.426
C06270=1196.303,323.405,-71.892,-176.403,7.685,148.426
C06271=1196.307,323.157,-71.860,-176.406,7.681,148.426
C06272=1196.311,322.909,-71.829,-176.408,7.679,148.426
C06273=1196.316,322.661,-71.798,-176.410,7.676,148.426
C06274=1196.319,322.413,-71.766,-176.413,7.673,148.426
C06275=1196.324,322.165,-71.736,-176.415,7.670,148.426
C06276=1196.328,321.917,-71.704,-176.417,7.667,148.426
C06277=1196.332,321.669,-71.673,-176.420,7.664,148.426
C06278=1196.336,321.421,-71.642,-176.422,7.661,148.426
C06279=1196.341,321.173,-71.610,-176.425,7.658,148.426
C06280=1196.345,320.925,-71.579,-176.427,7.656,148.426
C06281=1196.349,320.677,-71.549,-176.429,7.652,148.426
C06282=1196.353,320.430,-71.518,-176.432,7.649,148.426
C06283=1196.357,320.181,-71.486,-176.434,7.646,148.426
C06284=1196.362,319.933,-71.456,-176.436,7.644,148.425
C06285=1196.366,319.685,-71.425,-176.439,7.641,148.425
C06286=1196.370,319.437,-71.393,-176.442,7.638,148.425
C06287=1196.374,319.189,-71.362,-176.444,7.634,148.425
C06288=1196.378,318.941,-71.331,-176.446,7.632,148.425
C06289=1196.383,318.693,-71.300,-176.448,7.629,148.425
C06290=1196.386,318.445,-71.269,-176.451,7.626,148.425
C06291=1196.391,318.197,-71.238,-176.454,7.623,148.425
C06292=1196.395,317.949,-71.208,-176.456,7.621,148.425
C06293=1196.399,317.700,-71.177,-176.458,7.617,148.425
C06294=1196.404,317.452,-71.146,-176.461,7.614,148.425
C06295=1196.409,317.204,-71.115,-176.463,7.611,148.425
C06296=1196.411,316.957,-71.084,-176.465,7.609,148.425
C06297=1196.416,316.709,-71.053,-176.468,7.606,148.425
C06298=1196.421,316.461,-71.022,-176.470,7.603,148.425
C06299=1196.425,316.212,-70.991,-176.473,7.599,148.425
C06300=1196.429,315.964,-70.961,-176.475,7.597,148.425
C06301=1196.433,315.716,-70.930,-176.477,7.594,148.425
C06302=1196.437,315.468,-70.899,-176.480,7.591,148.424
C06303=1196.442,315.220,-70.868,-176.482,7.588,148.424
C06304=1196.447,314.944,-70.834,-176.485,7.585,148.424
C06305=1196.451,314.667,-70.800,-176.488,7.582,148.424
C06306=1196.456,314.391,-70.766,-176.490,7.579,148.424
C06307=1196.460,314.115,-70.731,-176.493,7.576,148.424
C06308=1196.465,313.867,-70.700,-176.495,7.573,148.424
C06309=1196.469,313.619,-70.670,-176.498,7.570,148.424
C06310=1196.473,313.371,-70.639,-176.500,7.567,148.424
C06311=1196.477,313.122,-70.608,-176.502,7.564,148.424
C06312=1196.482,312.874,-70.578,-176.505,7.561,148.424
C06313=1196.486,312.626,-70.548,-176.508,7.558,148.424
C06314=1196.491,312.378,-70.517,-176.510,7.556,148.424
C06315=1196.495,312.130,-70.486,-176.513,7.553,148.424
C06316=1196.498,311.882,-70.456,-176.515,7.549,148.424
C06317=1196.503,311.634,-70.425,-176.517,7.547,148.424
C06318=1196.507,311.386,-70.395,-176.520,7.544,148.424
C06319=1196.511,311.138,-70.364,-176.522,7.541,148.424
C06320=1196.516,310.889,-70.334,-176.525,7.538,148.424
C06321=1196.520,310.641,-70.304,-176.527,7.536,148.424
C06322=1196.524,310.393,-70.273,-176.529,7.533,148.424
C06323=1196.528,310.146,-70.243,-176.532,7.530,148.424
C06324=1196.532,309.897,-70.212,-176.535,7.527,148.424
C06325=1196.537,309.649,-70.182,-176.537,7.524,148.424
C06326=1196.541,309.401,-70.152,-176.539,7.521,148.424
C06327=1196.546,309.153,-70.121,-176.542,7.518,148.424
C06328=1196.550,308.905,-70.091,-176.544,7.516,148.424
C06329=1196.554,308.656,-70.060,-176.547,7.513,148.424
C06330=1196.558,308.408,-70.030,-176.549,7.510,148.424
C06331=1196.562,308.160,-69.999,-176.552,7.507,148.424
C06332=1196.567,307.912,-69.970,-176.554,7.504,148.424
C06333=1196.571,307.664,-69.939,-176.557,7.501,148.424
C06334=1196.575,307.417,-69.909,-176.559,7.498,148.424
C06335=1196.580,307.168,-69.879,-176.561,7.496,148.424
C06336=1196.583,306.920,-69.848,-176.564,7.493,148.424
C06337=1196.588,306.672,-69.817,-176.567,7.490,148.424
C06338=1196.592,306.423,-69.788,-176.569,7.487,148.424
C06339=1196.597,306.175,-69.757,-176.571,7.485,148.424
C06340=1196.601,305.927,-69.728,-176.574,7.482,148.424
C06341=1196.605,305.679,-69.697,-176.577,7.479,148.424
C06342=1196.610,305.431,-69.668,-176.579,7.476,148.424
C06343=1196.614,305.183,-69.637,-176.581,7.473,148.424
C06344=1196.617,304.935,-69.606,-176.584,7.470,148.424
C06345=1196.622,304.686,-69.577,-176.586,7.468,148.424
C06346=1196.626,304.438,-69.546,-176.588,7.465,148.424
C06347=1196.630,304.190,-69.517,-176.591,7.462,148.424
C06348=1196.635,303.942,-69.487,-176.594,7.459,148.424
C06349=1196.639,303.694,-69.456,-176.596,7.457,148.424
C06350=1196.643,303.446,-69.427,-176.599,7.454,148.424
C06351=1196.648,303.198,-69.396,-176.601,7.451,148.424
C06352=1196.652,302.949,-69.367,-176.604,7.448,148.424
C06353=1196.657,302.702,-69.336,-176.606,7.445,148.424
C06354=1196.661,302.453,-69.307,-176.609,7.442,148.424
C06355=1196.665,302.205,-69.277,-176.611,7.440,148.424
C06356=1196.670,301.957,-69.246,-176.614,7.437,148.424
C06357=1196.674,301.709,-69.217,-176.616,7.434,148.424
C06358=1196.678,301.461,-69.187,-176.618,7.432,148.424
C06359=1196.682,301.213,-69.157,-176.621,7.429,148.424
C06360=1196.686,300.964,-69.127,-176.624,7.426,148.424
C06361=1196.690,300.716,-69.097,-176.626,7.423,148.424
C06362=1196.694,300.468,-69.067,-176.628,7.420,148.424
C06363=1196.699,300.219,-69.037,-176.631,7.417,148.424
C06364=1196.704,299.971,-69.008,-176.633,7.415,148.424
C06365=1196.707,299.723,-68.978,-176.636,7.412,148.424
C06366=1196.712,299.475,-68.948,-176.639,7.409,148.424
C06367=1196.716,299.227,-68.919,-176.641,7.407,148.424
C06368=1196.721,298.978,-68.889,-176.643,7.404,148.424
C06369=1196.725,298.730,-68.858,-176.646,7.401,148.424
C06370=1196.729,298.482,-68.829,-176.649,7.398,148.424
C06371=1196.734,298.235,-68.800,-176.651,7.396,148.424
C06372=1196.738,297.986,-68.770,-176.654,7.393,148.424
C06373=1196.743,297.738,-68.740,-176.656,7.390,148.424
C06374=1196.747,297.489,-68.711,-176.659,7.388,148.424
C06375=1196.751,297.242,-68.681,-176.661,7.385,148.424
C06376=1196.755,296.994,-68.651,-176.664,7.382,148.424
C06377=1196.759,296.745,-68.622,-176.666,7.379,148.425
C06378=1196.763,296.497,-68.592,-176.669,7.376,148.425
C06379=1196.768,296.248,-68.562,-176.671,7.374,148.425
C06380=1196.772,296.000,-68.533,-176.674,7.371,148.425
C06381=1196.777,295.752,-68.503,-176.676,7.368,148.425
C06382=1196.781,295.504,-68.474,-176.678,7.366,148.425
C06383=1196.785,295.255,-68.445,-176.681,7.363,148.425
C06384=1196.789,295.007,-68.415,-176.684,7.360,148.425
C06385=1196.793,294.759,-68.386,-176.686,7.358,148.425
C06386=1196.797,294.511,-68.356,-176.689,7.355,148.425
C06387=1196.802,294.263,-68.327,-176.691,7.352,148.425
C06388=1196.806,294.015,-68.298,-176.694,7.350,148.425
C06389=1196.811,293.766,-68.268,-176.696,7.347,148.425
C06390=1196.815,293.518,-68.239,-176.699,7.344,148.425
C06391=1196.819,293.270,-68.209,-176.701,7.341,148.425
C06392=1196.824,293.021,-68.179,-176.704,7.338,148.425
C06393=1196.828,292.773,-68.150,-176.707,7.335,148.425
C06394=1196.832,292.525,-68.120,-176.709,7.333,148.425
C06395=1196.837,292.277,-68.091,-176.711,7.330,148.425
C06396=1196.841,292.029,-68.062,-176.713,7.328,148.425
C06397=1196.846,291.780,-68.033,-176.716,7.325,148.425
C06398=1196.849,291.532,-68.004,-176.719,7.322,148.425
C06399=1196.853,291.284,-67.975,-176.721,7.320,148.425
C06400=1196.857,291.036,-67.945,-176.724,7.317,148.425
C06401=1196.862,290.787,-67.916,-176.727,7.314,148.426
C06402=1196.866,290.540,-67.887,-176.729,7.312,148.426
C06403=1196.871,290.291,-67.858,-176.732,7.309,148.426
C06404=1196.875,290.043,-67.829,-176.734,7.306,148.426
C06405=1196.879,289.794,-67.799,-176.737,7.304,148.426
C06406=1196.883,289.546,-67.770,-176.739,7.301,148.426
C06407=1196.889,289.298,-67.741,-176.741,7.298,148.426
C06408=1196.892,289.023,-67.709,-176.744,7.295,148.426
C06409=1196.898,288.749,-67.676,-176.747,7.292,148.426
C06410=1196.903,288.474,-67.645,-176.750,7.290,148.426
C06411=1196.907,288.201,-67.612,-176.753,7.287,148.426
C06412=1196.912,287.952,-67.584,-176.755,7.284,148.426
C06413=1196.916,287.704,-67.554,-176.758,7.281,148.426
C06414=1196.920,287.455,-67.525,-176.760,7.279,148.426
C06415=1196.925,287.207,-67.496,-176.763,7.276,148.426
C06416=1196.929,286.959,-67.467,-176.765,7.273,148.426
C06417=1196.933,286.711,-67.438,-176.768,7.270,148.427
C06418=1196.937,286.462,-67.409,-176.771,7.268,148.427
C06419=1196.942,286.214,-67.380,-176.773,7.265,148.427
C06420=1196.947,285.965,-67.351,-176.776,7.262,148.427
C06421=1196.950,285.718,-67.323,-176.778,7.260,148.427
C06422=1196.955,285.469,-67.294,-176.781,7.257,148.427
C06423=1196.959,285.221,-67.265,-176.783,7.254,148.427
C06424=1196.964,284.972,-67.236,-176.786,7.252,148.427
C06425=1196.968,284.724,-67.207,-176.788,7.249,148.427
C06426=1196.972,284.476,-67.179,-176.791,7.247,148.427
C06427=1196.977,284.228,-67.149,-176.794,7.244,148.427
C06428=1196.981,283.979,-67.121,-176.796,7.241,148.427
C06429=1196.985,283.731,-67.091,-176.798,7.239,148.428
C06430=1196.990,283.483,-67.063,-176.801,7.236,148.428
C06431=1196.994,283.234,-67.034,-176.803,7.234,148.428
C06432=1196.998,282.986,-67.005,-176.806,7.231,148.428
C06433=1197.002,282.738,-66.977,-176.809,7.228,148.428
C06434=1197.007,282.489,-66.948,-176.811,7.226,148.428
C06435=1197.011,282.241,-66.919,-176.814,7.223,148.428
C06436=1197.015,281.993,-66.891,-176.816,7.221,148.428
C06437=1197.020,281.744,-66.862,-176.819,7.218,148.428
C06438=1197.025,281.496,-66.834,-176.821,7.216,148.428
C06439=1197.028,281.248,-66.805,-176.824,7.213,148.428
C06440=1197.033,280.999,-66.776,-176.827,7.210,148.428
C06441=1197.038,280.751,-66.748,-176.829,7.208,148.429
C06442=1197.041,280.503,-66.719,-176.832,7.205,148.429
C06443=1197.046,280.254,-66.690,-176.834,7.203,148.429
C06444=1197.050,280.006,-66.662,-176.837,7.200,148.429
C06445=1197.054,279.758,-66.633,-176.839,7.198,148.429
C06446=1197.059,279.509,-66.604,-176.842,7.195,148.429
C06447=1197.063,279.261,-66.576,-176.845,7.192,148.429
C06448=1197.068,279.013,-66.548,-176.847,7.189,148.429
C06449=1197.072,278.765,-66.520,-176.849,7.186,148.429
C06450=1197.076,278.516,-66.490,-176.852,7.185,148.429
C06451=1197.080,278.268,-66.462,-176.855,7.182,148.429
C06452=1197.085,278.020,-66.434,-176.857,7.179,148.430
C06453=1197.090,277.771,-66.405,-176.860,7.176,148.430
C06454=1197.094,277.523,-66.377,-176.862,7.174,148.430
C06455=1197.098,277.274,-66.349,-176.865,7.172,148.430
C06456=1197.102,277.027,-66.320,-176.867,7.169,148.430
C06457=1197.107,276.778,-66.291,-176.870,7.166,148.430
C06458=1197.111,276.530,-66.264,-176.873,7.163,148.430
C06459=1197.116,276.281,-66.235,-176.875,7.162,148.430
C06460=1197.120,276.033,-66.207,-176.878,7.158,148.430
C06461=1197.124,275.785,-66.179,-176.880,7.156,148.430
C06462=1197.128,275.536,-66.150,-176.883,7.153,148.430
C06463=1197.133,275.288,-66.122,-176.885,7.151,148.431
C06464=1197.137,275.039,-66.094,-176.888,7.148,148.431
C06465=1197.142,274.791,-66.066,-176.890,7.146,148.431
C06466=1197.146,274.542,-66.037,-176.893,7.143,148.431
C06467=1197.150,274.294,-66.009,-176.895,7.141,148.431
C06468=1197.155,274.045,-65.981,-176.898,7.138,148.431
C06469=1197.159,273.798,-65.953,-176.900,7.136,148.431
C06470=1197.163,273.549,-65.925,-176.903,7.133,148.431
C06471=1197.168,273.301,-65.896,-176.905,7.131,148.431
C06472=1197.172,273.052,-65.868,-176.908,7.128,148.432
C06473=1197.176,272.804,-65.840,-176.911,7.126,148.432
C06474=1197.181,272.555,-65.812,-176.913,7.123,148.432
C06475=1197.185,272.308,-65.784,-176.916,7.120,148.432
C06476=1197.189,272.059,-65.755,-176.919,7.118,148.432
C06477=1197.194,271.810,-65.728,-176.921,7.115,148.432
C06478=1197.198,271.562,-65.700,-176.923,7.113,148.432
C06479=1197.203,271.313,-65.672,-176.927,7.110,148.433
C06480=1197.207,271.066,-65.644,-176.929,7.108,148.433
C06481=1197.211,270.817,-65.616,-176.931,7.105,148.433
C06482=1197.215,270.569,-65.588,-176.934,7.103,148.433
C06483=1197.220,270.320,-65.560,-176.937,7.100,148.433
C06484=1197.225,270.072,-65.532,-176.939,7.098,148.433
C06485=1197.229,269.824,-65.504,-176.942,7.095,148.433
C06486=1197.233,269.575,-65.476,-176.944,7.093,148.433
C06487=1197.238,269.327,-65.448,-176.947,7.090,148.433
C06488=1197.242,269.078,-65.420,-176.949,7.088,148.434
C06489=1197.246,268.830,-65.393,-176.952,7.085,148.434
C06490=1197.251,268.582,-65.364,-176.954,7.083,148.434
C06491=1197.255,268.333,-65.337,-176.957,7.080,148.434
C06492=1197.260,268.085,-65.309,-176.959,7.078,148.434
C06493=1197.263,267.836,-65.281,-176.962,7.076,148.434
C06494=1197.269,267.587,-65.253,-176.965,7.073,148.434
C06495=1197.273,267.340,-65.225,-176.967,7.071,148.434
C06496=1197.277,267.091,-65.197,-176.970,7.068,148.434
C06497=1197.282,266.842,-65.170,-176.972,7.066,148.435
C06498=1197.286,266.595,-65.142,-176.975,7.063,148.435
C06499=1197.290,266.345,-65.115,-176.977,7.061,148.435
C06500=1197.295,266.097,-65.087,-176.980,7.058,148.435
C06501=1197.299,265.849,-65.059,-176.982,7.056,148.435
C06502=1197.303,265.600,-65.031,-176.985,7.053,148.435
C06503=1197.308,265.352,-65.004,-176.988,7.051,148.436
C06504=1197.312,265.104,-64.977,-176.990,7.048,148.436
C06505=1197.316,264.855,-64.948,-176.993,7.046,148.436
C06506=1197.321,264.607,-64.921,-176.996,7.044,148.436
C06507=1197.326,264.359,-64.893,-176.998,7.041,148.436
C06508=1197.330,264.109,-64.866,-177.001,7.038,148.436
C06509=1197.334,263.861,-64.838,-177.003,7.037,148.436
C06510=1197.339,263.613,-64.811,-177.005,7.034,148.437
C06511=1197.343,263.364,-64.783,-177.008,7.031,148.437
C06512=1197.348,263.092,-64.752,-177.011,7.029,148.437
C06513=1197.353,262.819,-64.723,-177.013,7.026,148.437
C06514=1197.358,262.545,-64.693,-177.017,7.024,148.437
C06515=1197.363,262.273,-64.662,-177.019,7.021,148.437
C06516=1197.367,262.025,-64.634,-177.022,7.019,148.438
C06517=1197.371,261.776,-64.607,-177.025,7.016,148.438
C06518=1197.376,261.527,-64.580,-177.027,7.014,148.438
C06519=1197.380,261.279,-64.552,-177.030,7.011,148.438
C06520=1197.385,261.031,-64.525,-177.032,7.009,148.438
C06521=1197.389,260.782,-64.498,-177.035,7.006,148.438
C06522=1197.393,260.534,-64.470,-177.037,7.004,148.438
C06523=1197.398,260.285,-64.443,-177.040,7.002,148.438
C06524=1197.403,260.037,-64.416,-177.043,6.999,148.439
C06525=1197.406,259.789,-64.389,-177.045,6.997,148.439
C06526=1197.410,259.540,-64.361,-177.048,6.994,148.439
C06527=1197.415,259.292,-64.334,-177.050,6.992,148.439
C06528=1197.420,259.043,-64.307,-177.053,6.989,148.439
C06529=1197.424,258.795,-64.279,-177.056,6.987,148.439
C06530=1197.429,258.547,-64.252,-177.058,6.985,148.440
C06531=1197.433,258.298,-64.225,-177.061,6.982,148.440
C06532=1197.437,258.049,-64.198,-177.063,6.980,148.440
C06533=1197.442,257.801,-64.170,-177.066,6.977,148.440
C06534=1197.446,257.553,-64.143,-177.068,6.976,148.440
C06535=1197.451,257.304,-64.116,-177.071,6.973,148.440
C06536=1197.455,257.055,-64.088,-177.073,6.970,148.440
C06537=1197.459,256.807,-64.062,-177.076,6.968,148.441
C06538=1197.464,256.558,-64.035,-177.079,6.965,148.441
C06539=1197.468,256.310,-64.008,-177.081,6.964,148.441
C06540=1197.473,256.061,-63.981,-177.084,6.961,148.441
C06541=1197.477,255.813,-63.953,-177.087,6.959,148.441
C06542=1197.482,255.565,-63.926,-177.089,6.957,148.442
C06543=1197.485,255.316,-63.899,-177.092,6.954,148.442
C06544=1197.490,255.068,-63.872,-177.094,6.952,148.442
C06545=1197.495,254.819,-63.845,-177.097,6.949,148.442
C06546=1197.499,254.571,-63.818,-177.099,6.947,148.442
C06547=1197.504,254.322,-63.791,-177.102,6.945,148.442
C06548=1197.508,254.074,-63.764,-177.105,6.942,148.443
C06549=1197.512,253.825,-63.737,-177.107,6.940,148.443
C06550=1197.517,253.577,-63.710,-177.109,6.938,148.443
C06551=1197.521,253.328,-63.683,-177.112,6.935,148.443
C06552=1197.525,253.080,-63.656,-177.114,6.933,148.443
C06553=1197.530,252.831,-63.629,-177.118,6.930,148.443
C06554=1197.534,252.583,-63.602,-177.120,6.928,148.444
C06555=1197.539,252.334,-63.575,-177.122,6.926,148.444
C06556=1197.543,252.085,-63.549,-177.125,6.923,148.444
C06557=1197.548,251.837,-63.522,-177.128,6.921,148.444
C06558=1197.553,251.588,-63.495,-177.130,6.919,148.444
C06559=1197.556,251.340,-63.469,-177.133,6.916,148.444
C06560=1197.561,251.092,-63.442,-177.135,6.914,148.445
C06561=1197.566,250.843,-63.415,-177.138,6.911,148.445
C06562=1197.570,250.595,-63.388,-177.141,6.910,148.445
C06563=1197.575,250.346,-63.362,-177.143,6.907,148.445
C06564=1197.579,250.097,-63.335,-177.146,6.905,148.445
C06565=1197.583,249.849,-63.308,-177.148,6.903,148.445
C06566=1197.588,249.601,-63.281,-177.151,6.901,148.446
C06567=1197.593,249.352,-63.254,-177.153,6.898,148.446
C06568=1197.597,249.103,-63.229,-177.156,6.896,148.446
C06569=1197.601,248.855,-63.201,-177.158,6.894,148.446
C06570=1197.605,248.606,-63.175,-177.161,6.891,148.447
C06571=1197.609,248.357,-63.148,-177.164,6.889,148.447
C06572=1197.614,248.108,-63.121,-177.166,6.887,148.447
C06573=1197.619,247.861,-63.095,-177.169,6.884,148.447
C06574=1197.624,247.612,-63.068,-177.172,6.882,148.447
C06575=1197.628,247.364,-63.042,-177.174,6.880,148.447
C06576=1197.632,247.115,-63.015,-177.177,6.877,148.448
C06577=1197.637,246.867,-62.988,-177.179,6.875,148.448
C06578=1197.641,246.618,-62.962,-177.182,6.873,148.448
C06579=1197.646,246.369,-62.935,-177.184,6.870,148.448
C06580=1197.650,246.121,-62.909,-177.187,6.868,148.448
C06581=1197.655,245.872,-62.883,-177.189,6.866,148.449
C06582=1197.659,245.624,-62.856,-177.192,6.864,148.449
C06583=1197.663,245.375,-62.829,-177.195,6.861,148.449
C06584=1197.668,245.126,-62.803,-177.197,6.860,148.449
C06585=1197.672,244.878,-62.776,-177.200,6.857,148.449
C06586=1197.677,244.629,-62.750,-177.203,6.855,148.450
C06587=1197.681,244.381,-62.723,-177.205,6.853,148.450
C06588=1197.685,244.132,-62.698,-177.208,6.850,148.450
C06589=1197.689,243.884,-62.671,-177.210,6.848,148.450
C06590=1197.694,243.635,-62.645,-177.213,6.846,148.450
C06591=1197.698,243.386,-62.618,-177.215,6.843,148.450
C06592=1197.704,243.138,-62.592,-177.218,6.841,148.451
C06593=1197.708,242.890,-62.566,-177.220,6.839,148.451
C06594=1197.713,242.641,-62.540,-177.223,6.836,148.451
C06595=1197.717,242.392,-62.513,-177.226,6.834,148.451
C06596=1197.721,242.144,-62.487,-177.228,6.832,148.452
C06597=1197.725,241.895,-62.460,-177.231,6.830,148.452
C06598=1197.730,241.646,-62.435,-177.234,6.827,148.452
C06599=1197.735,241.397,-62.408,-177.236,6.826,148.452
C06600=1197.739,241.149,-62.382,-177.238,6.823,148.452
C06601=1197.743,240.901,-62.356,-177.242,6.821,148.453
C06602=1197.748,240.652,-62.330,-177.244,6.819,148.453
C06603=1197.752,240.404,-62.304,-177.246,6.817,148.453
C06604=1197.757,240.155,-62.278,-177.250,6.814,148.453
C06605=1197.761,239.906,-62.251,-177.252,6.812,148.453
C06606=1197.765,239.658,-62.225,-177.254,6.810,148.454
C06607=1197.770,239.409,-62.200,-177.257,6.808,148.454
C06608=1197.775,239.160,-62.173,-177.260,6.805,148.454
C06609=1197.779,238.912,-62.147,-177.262,6.803,148.454
C06610=1197.783,238.663,-62.121,-177.264,6.801,148.455
C06611=1197.788,238.414,-62.095,-177.267,6.799,148.455
C06612=1197.793,238.165,-62.069,-177.270,6.796,148.455
C06613=1197.797,237.918,-62.043,-177.272,6.795,148.455
C06614=1197.801,237.669,-62.017,-177.275,6.792,148.455
C06615=1197.806,237.420,-61.991,-177.278,6.790,148.456
C06616=1197.811,237.149,-61.962,-177.280,6.788,148.456
C06617=1197.816,236.878,-61.934,-177.283,6.785,148.456
C06618=1197.821,236.606,-61.906,-177.286,6.783,148.456
C06619=1197.825,236.334,-61.878,-177.289,6.780,148.457
C06620=1197.831,236.086,-61.852,-177.291,6.778,148.457
C06621=1197.835,235.837,-61.826,-177.294,6.776,148.457
C06622=1197.839,235.588,-61.800,-177.297,6.774,148.457
C06623=1197.843,235.339,-61.774,-177.299,6.772,148.457
C06624=1197.848,235.091,-61.749,-177.302,6.770,148.458
C06625=1197.853,234.843,-61.722,-177.304,6.768,148.458
C06626=1197.857,234.594,-61.696,-177.307,6.765,148.458
C06627=1197.861,234.345,-61.670,-177.310,6.763,148.458
C06628=1197.866,234.097,-61.645,-177.312,6.761,148.459
C06629=1197.870,233.848,-61.619,-177.315,6.759,148.459
C06630=1197.874,233.600,-61.593,-177.318,6.756,148.459
C06631=1197.879,233.351,-61.568,-177.320,6.754,148.459
C06632=1197.884,233.102,-61.542,-177.323,6.752,148.460
C06633=1197.888,232.854,-61.516,-177.325,6.750,148.460
C06634=1197.893,232.605,-61.490,-177.328,6.748,148.460
C06635=1197.897,232.357,-61.465,-177.331,6.746,148.460
C06636=1197.902,232.108,-61.439,-177.333,6.744,148.460
C06637=1197.906,231.859,-61.413,-177.335,6.742,148.461
C06638=1197.911,231.611,-61.388,-177.339,6.739,148.461
C06639=1197.915,231.362,-61.362,-177.341,6.737,148.461
C06640=1197.919,231.113,-61.336,-177.343,6.735,148.461
C06641=1197.924,230.865,-61.312,-177.346,6.733,148.462
C06642=1197.929,230.616,-61.286,-177.348,6.731,148.462
C06643=1197.933,230.367,-61.260,-177.351,6.728,148.462
C06644=1197.938,230.119,-61.235,-177.354,6.727,148.463
C06645=1197.943,229.870,-61.209,-177.356,6.725,148.463
C06646=1197.947,229.621,-61.183,-177.359,6.723,148.463
C06647=1197.952,229.373,-61.157,-177.362,6.720,148.463
C06648=1197.956,229.123,-61.132,-177.364,6.718,148.463
C06649=1197.960,228.875,-61.107,-177.367,6.716,148.464
C06650=1197.965,228.627,-61.081,-177.370,6.714,148.464
C06651=1197.969,228.378,-61.056,-177.372,6.712,148.464
C06652=1197.973,228.129,-61.030,-177.375,6.709,148.464
C06653=1197.978,227.881,-61.006,-177.378,6.708,148.465
C06654=1197.982,227.632,-60.980,-177.380,6.705,148.465
C06655=1197.987,227.384,-60.955,-177.382,6.704,148.465
C06656=1197.991,227.135,-60.929,-177.386,6.701,148.465
C06657=1197.996,226.885,-60.904,-177.388,6.699,148.466
C06658=1198.001,226.637,-60.878,-177.390,6.697,148.466
C06659=1198.005,226.388,-60.853,-177.393,6.695,148.466
C06660=1198.010,226.140,-60.827,-177.395,6.693,148.466
C06661=1198.014,225.891,-60.802,-177.398,6.690,148.467
C06662=1198.019,225.643,-60.777,-177.401,6.688,148.467
C06663=1198.023,225.394,-60.751,-177.403,6.686,148.467
C06664=1198.027,225.145,-60.727,-177.406,6.684,148.467
C06665=1198.032,224.897,-60.701,-177.408,6.683,148.468
C06666=1198.036,224.647,-60.676,-177.412,6.680,148.468
C06667=1198.041,224.399,-60.651,-177.414,6.678,148.468
C06668=1198.046,224.150,-60.625,-177.416,6.676,148.468
C06669=1198.051,223.902,-60.600,-177.419,6.674,148.469
C06670=1198.055,223.653,-60.575,-177.421,6.672,148.469
C06671=1198.059,223.405,-60.551,-177.424,6.670,148.469
C06672=1198.063,223.156,-60.525,-177.427,6.667,148.470
C06673=1198.069,222.907,-60.500,-177.430,6.666,148.470
C06674=1198.073,222.658,-60.474,-177.432,6.663,148.470
C06675=1198.078,222.409,-60.450,-177.435,6.662,148.470
C06676=1198.081,222.161,-60.425,-177.437,6.660,148.471
C06677=1198.087,221.912,-60.400,-177.440,6.657,148.471
C06678=1198.091,221.663,-60.374,-177.443,6.655,148.471
C06679=1198.096,221.415,-60.349,-177.445,6.653,148.471
C06680=1198.099,221.166,-60.324,-177.448,6.651,148.472
C06681=1198.105,220.918,-60.300,-177.450,6.649,148.472
C06682=1198.109,220.669,-60.274,-177.453,6.647,148.472
C06683=1198.114,220.420,-60.249,-177.456,6.645,148.472
C06684=1198.117,220.172,-60.224,-177.459,6.643,148.473
C06685=1198.123,219.923,-60.199,-177.461,6.641,148.473
C06686=1198.127,219.673,-60.174,-177.463,6.639,148.473
C06687=1198.132,219.425,-60.149,-177.466,6.637,148.474
C06688=1198.136,219.176,-60.125,-177.469,6.635,148.474
C06689=1198.141,218.927,-60.100,-177.471,6.632,148.474
C06690=1198.145,218.679,-60.074,-177.474,6.630,148.474
C06691=1198.149,218.430,-60.050,-177.477,6.629,148.475
C06692=1198.155,218.181,-60.025,-177.479,6.627,148.475
C06693=1198.159,217.933,-60.000,-177.481,6.625,148.475
C06694=1198.163,217.684,-59.976,-177.484,6.623,148.475
C06695=1198.168,217.435,-59.951,-177.487,6.620,148.476
C06696=1198.172,217.187,-59.926,-177.490,6.618,148.476
C06697=1198.177,216.938,-59.901,-177.493,6.617,148.476
C06698=1198.181,216.689,-59.876,-177.495,6.614,148.476
C06699=1198.186,216.440,-59.852,-177.497,6.613,148.477
C06700=1198.190,216.192,-59.826,-177.500,6.611,148.477
C06701=1198.195,215.943,-59.802,-177.503,6.608,148.477
C06702=1198.200,215.695,-59.777,-177.505,6.606,148.478
C06703=1198.204,215.445,-59.752,-177.508,6.604,148.478
C06704=1198.209,215.197,-59.728,-177.511,6.602,148.478
C06705=1198.213,214.948,-59.703,-177.513,6.600,148.479
C06706=1198.217,214.699,-59.679,-177.516,6.599,148.479
C06707=1198.222,214.451,-59.654,-177.518,6.596,148.479
C06708=1198.226,214.202,-59.629,-177.521,6.594,148.479
C06709=1198.231,213.953,-59.605,-177.524,6.592,148.480
C06710=1198.236,213.704,-59.580,-177.527,6.590,148.480
C06711=1198.240,213.455,-59.556,-177.529,6.588,148.480
C06712=1198.245,213.206,-59.531,-177.532,6.586,148.480
C06713=1198.249,212.959,-59.506,-177.534,6.584,148.481
C06714=1198.254,212.709,-59.481,-177.537,6.583,148.481
C06715=1198.258,212.461,-59.457,-177.540,6.580,148.481
C06716=1198.263,212.212,-59.432,-177.543,6.578,148.482
C06717=1198.267,211.963,-59.408,-177.545,6.576,148.482
C06718=1198.272,211.714,-59.384,-177.547,6.574,148.482
C06719=1198.277,211.466,-59.359,-177.550,6.572,148.483
C06720=1198.282,211.196,-59.333,-177.553,6.570,148.483
C06721=1198.287,210.924,-59.306,-177.556,6.568,148.483
C06722=1198.291,210.654,-59.280,-177.559,6.566,148.483
C06723=1198.296,210.384,-59.253,-177.562,6.563,148.484
C06724=1198.301,210.135,-59.229,-177.565,6.562,148.484
C06725=1198.305,209.886,-59.204,-177.567,6.560,148.484
C06726=1198.310,209.638,-59.180,-177.570,6.558,148.485
C06727=1198.315,209.389,-59.155,-177.572,6.556,148.485
C06728=1198.319,209.140,-59.131,-177.575,6.554,148.485
C06729=1198.324,208.891,-59.106,-177.577,6.552,148.486
C06730=1198.328,208.642,-59.083,-177.580,6.550,148.486
C06731=1198.333,208.394,-59.059,-177.583,6.548,148.486
C06732=1198.338,208.145,-59.034,-177.586,6.546,148.487
C06733=1198.342,207.896,-59.010,-177.588,6.544,148.487
C06734=1198.347,207.647,-58.985,-177.591,6.542,148.487
C06735=1198.351,207.399,-58.961,-177.593,6.540,148.487
C06736=1198.356,207.150,-58.938,-177.596,6.538,148.488
C06737=1198.360,206.900,-58.913,-177.599,6.536,148.488
C06738=1198.365,206.652,-58.889,-177.601,6.535,148.488
C06739=1198.369,206.404,-58.865,-177.603,6.532,148.489
C06740=1198.374,206.155,-58.840,-177.606,6.531,148.489
C06741=1198.379,205.906,-58.817,-177.609,6.529,148.489
C06742=1198.383,205.657,-58.792,-177.611,6.527,148.490
C06743=1198.387,205.408,-58.768,-177.614,6.525,148.490
C06744=1198.392,205.160,-58.743,-177.617,6.522,148.490
C06745=1198.397,204.911,-58.720,-177.620,6.521,148.491
C06746=1198.402,204.662,-58.696,-177.622,6.518,148.491
C06747=1198.406,204.414,-58.672,-177.625,6.517,148.491
C06748=1198.411,204.164,-58.647,-177.627,6.515,148.491
C06749=1198.415,203.915,-58.623,-177.630,6.513,148.492
C06750=1198.420,203.667,-58.599,-177.633,6.511,148.492
C06751=1198.424,203.418,-58.576,-177.635,6.509,148.492
C06752=1198.429,203.169,-58.552,-177.638,6.508,148.493
C06753=1198.434,202.921,-58.527,-177.641,6.506,148.493
C06754=1198.438,202.671,-58.504,-177.643,6.504,148.493
C06755=1198.442,202.423,-58.479,-177.645,6.502,148.494
C06756=1198.447,202.173,-58.456,-177.648,6.500,148.494
C06757=1198.451,201.925,-58.432,-177.651,6.498,148.494
C06758=1198.456,201.677,-58.408,-177.654,6.496,148.495
C06759=1198.461,201.427,-58.384,-177.657,6.494,148.495
C06760=1198.466,201.179,-58.360,-177.659,6.492,148.495
C06761=1198.470,200.930,-58.337,-177.662,6.490,148.496
C06762=1198.474,200.681,-58.312,-177.664,6.488,148.496
C06763=1198.479,200.432,-58.289,-177.667,6.486,148.496
C06764=1198.483,200.183,-58.265,-177.669,6.484,148.496
C06765=1198.488,199.934,-58.241,-177.672,6.482,148.497
C06766=1198.493,199.686,-58.217,-177.675,6.481,148.497
C06767=1198.498,199.437,-58.193,-177.677,6.479,148.497
C06768=1198.502,199.188,-58.169,-177.680,6.477,148.498
C06769=1198.507,198.939,-58.146,-177.683,6.475,148.498
C06770=1198.511,198.691,-58.122,-177.685,6.473,148.498
C06771=1198.516,198.442,-58.098,-177.688,6.472,148.499
C06772=1198.521,198.193,-58.075,-177.690,6.469,148.499
C06773=1198.525,197.944,-58.051,-177.693,6.468,148.499
C06774=1198.530,197.695,-58.028,-177.695,6.466,148.500
C06775=1198.534,197.447,-58.004,-177.698,6.464,148.500
C06776=1198.539,197.198,-57.980,-177.701,6.462,148.500
C06777=1198.543,196.949,-57.957,-177.703,6.460,148.501
C06778=1198.548,196.700,-57.933,-177.706,6.459,148.501
C06779=1198.552,196.451,-57.909,-177.709,6.457,148.501
C06780=1198.557,196.201,-57.886,-177.711,6.455,148.502
C06781=1198.561,195.953,-57.862,-177.714,6.453,148.502
C06782=1198.566,195.704,-57.838,-177.717,6.451,148.502
C06783=1198.570,195.455,-57.815,-177.719,6.450,148.503
C06784=1198.575,195.206,-57.792,-177.722,6.448,148.503
C06785=1198.580,194.958,-57.767,-177.724,6.446,148.503
C06786=1198.584,194.709,-57.744,-177.727,6.444,148.504
C06787=1198.590,194.460,-57.721,-177.730,6.442,148.504
C06788=1198.594,194.211,-57.698,-177.732,6.440,148.504
C06789=1198.599,193.963,-57.674,-177.735,6.438,148.505
C06790=1198.603,193.714,-57.650,-177.737,6.436,148.505
C06791=1198.608,193.465,-57.627,-177.740,6.435,148.505
C06792=1198.613,193.216,-57.604,-177.743,6.433,148.506
C06793=1198.617,192.967,-57.580,-177.745,6.431,148.506
C06794=1198.621,192.719,-57.557,-177.748,6.429,148.506
C06795=1198.626,192.470,-57.533,-177.751,6.427,148.507
C06796=1198.630,192.220,-57.510,-177.753,6.426,148.507
C06797=1198.635,191.971,-57.487,-177.756,6.424,148.507
C06798=1198.640,191.722,-57.463,-177.759,6.422,148.508
C06799=1198.645,191.473,-57.440,-177.761,6.420,148.508
C06800=1198.649,191.224,-57.417,-177.764,6.418,148.508
C06801=1198.653,190.976,-57.394,-177.767,6.417,148.509
C06802=1198.658,190.727,-57.370,-177.769,6.415,148.509
C06803=1198.662,190.478,-57.346,-177.772,6.413,148.509
C06804=1198.668,190.230,-57.323,-177.774,6.411,148.510
C06805=1198.672,189.981,-57.300,-177.777,6.409,148.510
C06806=1198.677,189.732,-57.277,-177.780,6.407,148.510
C06807=1198.681,189.483,-57.254,-177.782,6.405,148.511
C06808=1198.686,189.234,-57.231,-177.785,6.404,148.511
C06809=1198.690,188.985,-57.207,-177.788,6.402,148.511
C06810=1198.695,188.736,-57.184,-177.790,6.400,148.512
C06811=1198.700,188.487,-57.160,-177.793,6.398,148.512
C06812=1198.704,188.239,-57.138,-177.795,6.396,148.512
C06813=1198.709,187.990,-57.115,-177.798,6.395,148.513
C06814=1198.714,187.741,-57.091,-177.801,6.393,148.513
C06815=1198.718,187.492,-57.068,-177.803,6.391,148.513
C06816=1198.722,187.243,-57.045,-177.806,6.389,148.514
C06817=1198.727,186.993,-57.023,-177.809,6.387,148.514
C06818=1198.732,186.744,-56.999,-177.811,6.386,148.515
C06819=1198.737,186.496,-56.977,-177.814,6.384,148.515
C06820=1198.741,186.247,-56.953,-177.817,6.382,148.515
C06821=1198.746,185.998,-56.930,-177.819,6.380,148.516
C06822=1198.751,185.749,-56.907,-177.822,6.378,148.516
C06823=1198.755,185.501,-56.884,-177.824,6.377,148.516
C06824=1198.760,185.231,-56.859,-177.827,6.375,148.517
C06825=1198.765,184.961,-56.835,-177.830,6.373,148.517
C06826=1198.770,184.692,-56.810,-177.833,6.371,148.518
C06827=1198.775,184.422,-56.784,-177.836,6.370,148.518
C06828=1198.779,184.173,-56.762,-177.839,6.368,148.518
C06829=1198.785,183.925,-56.739,-177.841,6.366,148.519
C06830=1198.790,183.675,-56.716,-177.844,6.364,148.519
C06831=1198.794,183.426,-56.693,-177.847,6.362,148.519
C06832=1198.798,183.177,-56.670,-177.849,6.361,148.520
C06833=1198.803,182.929,-56.648,-177.852,6.359,148.520
C06834=1198.808,182.680,-56.625,-177.855,6.357,148.520
C06835=1198.812,182.431,-56.602,-177.857,6.355,148.521
C06836=1198.816,182.182,-56.579,-177.860,6.353,148.521
C06837=1198.821,181.933,-56.555,-177.862,6.352,148.522
C06838=1198.826,181.684,-56.534,-177.865,6.351,148.522
C06839=1198.831,181.435,-56.510,-177.867,6.349,148.522
C06840=1198.835,181.187,-56.488,-177.870,6.347,148.523
C06841=1198.840,180.937,-56.465,-177.873,6.345,148.523
C06842=1198.845,180.689,-56.442,-177.875,6.343,148.523
C06843=1198.849,180.439,-56.420,-177.878,6.342,148.524
C06844=1198.854,180.190,-56.397,-177.881,6.340,148.524
C06845=1198.859,179.942,-56.374,-177.883,6.338,148.524
C06846=1198.864,179.692,-56.352,-177.886,6.336,148.525
C06847=1198.867,179.444,-56.329,-177.889,6.334,148.525
C06848=1198.873,179.194,-56.306,-177.891,6.333,148.525
C06849=1198.877,178.946,-56.284,-177.893,6.332,148.526
C06850=1198.882,178.697,-56.260,-177.896,6.330,148.526
C06851=1198.886,178.448,-56.238,-177.899,6.328,148.527
C06852=1198.891,178.200,-56.216,-177.901,6.326,148.527
C06853=1198.896,177.950,-56.193,-177.904,6.324,148.527
C06854=1198.900,177.701,-56.171,-177.907,6.323,148.528
C06855=1198.905,177.452,-56.148,-177.909,6.321,148.528
C06856=1198.909,177.204,-56.125,-177.912,6.319,148.529
C06857=1198.914,176.954,-56.103,-177.915,6.317,148.529
C06858=1198.919,176.706,-56.080,-177.917,6.317,148.529
C06859=1198.924,176.456,-56.058,-177.920,6.315,148.530
C06860=1198.928,176.208,-56.035,-177.923,6.313,148.530
C06861=1198.933,175.959,-56.013,-177.925,6.311,148.530
C06862=1198.938,175.709,-55.991,-177.928,6.309,148.531
C06863=1198.942,175.461,-55.968,-177.931,6.308,148.531
C06864=1198.947,175.212,-55.946,-177.933,6.306,148.531
C06865=1198.951,174.963,-55.923,-177.936,6.304,148.532
C06866=1198.956,174.714,-55.901,-177.938,6.303,148.532
C06867=1198.961,174.465,-55.879,-177.941,6.301,148.533
C06868=1198.965,174.216,-55.856,-177.943,6.299,148.533
C06869=1198.970,173.967,-55.834,-177.946,6.298,148.533
C06870=1198.975,173.718,-55.811,-177.949,6.296,148.534
C06871=1198.979,173.470,-55.789,-177.952,6.294,148.534
C06872=1198.984,173.220,-55.767,-177.954,6.292,148.535
C06873=1198.989,172.971,-55.744,-177.957,6.291,148.535
C06874=1198.993,172.723,-55.722,-177.959,6.290,148.535
C06875=1198.997,172.473,-55.700,-177.962,6.288,148.536
C06876=1199.003,172.224,-55.678,-177.965,6.286,148.536
C06877=1199.007,171.975,-55.656,-177.967,6.284,148.536
C06878=1199.012,171.727,-55.633,-177.970,6.283,148.537
C06879=1199.016,171.478,-55.611,-177.973,6.281,148.537
C06880=1199.021,171.228,-55.589,-177.975,6.279,148.538
C06881=1199.026,170.979,-55.567,-177.977,6.278,148.538
C06882=1199.030,170.731,-55.544,-177.980,6.276,148.538
C06883=1199.035,170.482,-55.522,-177.983,6.275,148.539
C06884=1199.040,170.232,-55.500,-177.986,6.273,148.539
C06885=1199.045,169.984,-55.478,-177.989,6.271,148.540
C06886=1199.049,169.734,-55.456,-177.991,6.269,148.540
C06887=1199.054,169.486,-55.434,-177.993,6.268,148.540
C06888=1199.059,169.237,-55.411,-177.996,6.267,148.541
C06889=1199.063,168.988,-55.389,-177.999,6.265,148.541
C06890=1199.068,168.739,-55.367,-178.001,6.263,148.541
C06891=1199.073,168.490,-55.346,-178.004,6.261,148.542
C06892=1199.077,168.241,-55.324,-178.007,6.259,148.542
C06893=1199.082,167.992,-55.301,-178.009,6.259,148.543
C06894=1199.087,167.742,-55.279,-178.012,6.257,148.543
C06895=1199.092,167.494,-55.258,-178.015,6.255,148.544
C06896=1199.096,167.244,-55.235,-178.017,6.253,148.544
C06897=1199.100,166.996,-55.213,-178.020,6.252,148.544
C06898=1199.105,166.747,-55.191,-178.023,6.250,148.545
C06899=1199.110,166.498,-55.169,-178.025,6.249,148.545
C06900=1199.115,166.249,-55.147,-178.027,6.247,148.545
C06901=1199.119,166.000,-55.125,-178.031,6.246,148.546
C06902=1199.124,165.751,-55.103,-178.033,6.244,148.546
C06903=1199.129,165.502,-55.081,-178.036,6.242,148.547
C06904=1199.133,165.253,-55.059,-178.038,6.241,148.547
C06905=1199.138,165.004,-55.038,-178.041,6.239,148.547
C06906=1199.143,164.755,-55.016,-178.043,6.237,148.548
C06907=1199.147,164.506,-54.995,-178.046,6.236,148.548
C06908=1199.152,164.257,-54.973,-178.049,6.234,148.549
C06909=1199.156,164.008,-54.951,-178.051,6.233,148.549
C06910=1199.161,163.759,-54.929,-178.054,6.231,148.550
C06911=1199.165,163.510,-54.907,-178.057,6.230,148.550
C06912=1199.170,163.261,-54.885,-178.059,6.228,148.550
C06913=1199.175,163.012,-54.864,-178.062,6.226,148.551
C06914=1199.179,162.763,-54.842,-178.064,6.225,148.551
C06915=1199.184,162.514,-54.820,-178.067,6.223,148.551
C06916=1199.189,162.265,-54.798,-178.070,6.222,148.552
C06917=1199.194,162.016,-54.777,-178.073,6.220,148.552
C06918=1199.199,161.767,-54.755,-178.075,6.218,148.553
C06919=1199.203,161.518,-54.733,-178.077,6.217,148.553
C06920=1199.208,161.269,-54.712,-178.080,6.215,148.554
C06921=1199.212,161.020,-54.690,-178.083,6.214,148.554
C06922=1199.217,160.770,-54.669,-178.086,6.212,148.554
C06923=1199.222,160.522,-54.647,-178.088,6.211,148.555
C06924=1199.226,160.272,-54.625,-178.091,6.209,148.555
C06925=1199.231,160.024,-54.603,-178.093,6.208,148.556
C06926=1199.236,159.775,-54.582,-178.096,6.206,148.556
C06927=1199.241,159.525,-54.560,-178.099,6.204,148.556
C06928=1199.246,159.257,-54.536,-178.102,6.203,148.557
C06929=1199.251,158.987,-54.513,-178.104,6.201,148.557
C06930=1199.256,158.718,-54.490,-178.107,6.199,148.558
C06931=1199.261,158.449,-54.467,-178.110,6.198,148.558
C06932=1199.266,158.200,-54.445,-178.112,6.197,148.559
C06933=1199.271,157.952,-54.424,-178.115,6.195,148.559
C06934=1199.276,157.703,-54.403,-178.118,6.193,148.559
C06935=1199.280,157.453,-54.381,-178.120,6.191,148.560
C06936=1199.285,157.205,-54.359,-178.123,6.191,148.560
C06937=1199.289,156.956,-54.339,-178.126,6.189,148.561
C06938=1199.294,156.706,-54.317,-178.128,6.187,148.561
C06939=1199.298,156.458,-54.295,-178.131,6.185,148.562
C06940=1199.304,156.208,-54.274,-178.133,6.184,148.562
C06941=1199.308,155.960,-54.252,-178.136,6.183,148.563
C06942=1199.313,155.710,-54.231,-178.139,6.181,148.563
C06943=1199.317,155.461,-54.210,-178.142,6.179,148.563
C06944=1199.322,155.212,-54.189,-178.144,6.178,148.564
C06945=1199.327,154.963,-54.167,-178.146,6.177,148.564
C06946=1199.332,154.714,-54.146,-178.150,6.175,148.565
C06947=1199.337,154.465,-54.124,-178.152,6.173,148.565
C06948=1199.341,154.216,-54.104,-178.154,6.172,148.565
C06949=1199.345,153.967,-54.082,-178.157,6.171,148.566
C06950=1199.351,153.717,-54.061,-178.160,6.169,148.566
C06951=1199.355,153.469,-54.039,-178.162,6.168,148.567
C06952=1199.360,153.220,-54.019,-178.165,6.166,148.567
C06953=1199.365,152.971,-53.997,-178.168,6.165,148.568
C06954=1199.369,152.721,-53.976,-178.170,6.163,148.568
C06955=1199.374,152.473,-53.954,-178.172,6.162,148.568
C06956=1199.379,152.224,-53.934,-178.176,6.160,148.569
C06957=1199.383,151.975,-53.912,-178.178,6.159,148.569
C06958=1199.388,151.725,-53.891,-178.181,6.157,148.570
C06959=1199.393,151.476,-53.870,-178.183,6.156,148.570
C06960=1199.397,151.227,-53.849,-178.186,6.154,148.571
C06961=1199.403,150.978,-53.828,-178.189,6.153,148.571
C06962=1199.407,150.729,-53.806,-178.191,6.152,148.571
C06963=1199.412,150.481,-53.786,-178.194,6.150,148.572
C06964=1199.416,150.231,-53.764,-178.196,6.148,148.572
C06965=1199.421,149.982,-53.743,-178.200,6.147,148.573
C06966=1199.426,149.733,-53.722,-178.202,6.146,148.573
C06967=1199.431,149.484,-53.701,-178.204,6.144,148.574
C06968=1199.436,149.235,-53.680,-178.207,6.142,148.574
C06969=1199.440,148.986,-53.659,-178.210,6.142,148.575
C06970=1199.445,148.736,-53.638,-178.212,6.140,148.575
C06971=1199.449,148.487,-53.618,-178.215,6.138,148.575
C06972=1199.454,148.239,-53.596,-178.217,6.137,148.576
C06973=1199.459,147.989,-53.575,-178.220,6.136,148.576
C06974=1199.464,147.740,-53.555,-178.223,6.134,148.577
C06975=1199.469,147.491,-53.534,-178.226,6.132,148.577
C06976=1199.473,147.243,-53.512,-178.228,6.131,148.577
C06977=1199.478,146.993,-53.491,-178.231,6.130,148.578
C06978=1199.483,146.744,-53.470,-178.234,6.128,148.578
C06979=1199.487,146.495,-53.450,-178.236,6.127,148.579
C06980=1199.492,146.245,-53.429,-178.238,6.125,148.579
C06981=1199.496,145.997,-53.408,-178.242,6.124,148.580
C06982=1199.502,145.748,-53.387,-178.244,6.123,148.580
C06983=1199.506,145.499,-53.366,-178.246,6.121,148.581
C06984=1199.511,145.250,-53.345,-178.249,6.119,148.581
C06985=1199.516,145.001,-53.325,-178.252,6.119,148.582
C06986=1199.521,144.751,-53.304,-178.254,6.117,148.582
C06987=1199.525,144.502,-53.283,-178.257,6.115,148.582
C06988=1199.530,144.253,-53.262,-178.259,6.114,148.583
C06989=1199.534,144.004,-53.241,-178.262,6.113,148.583
C06990=1199.539,143.755,-53.220,-178.265,6.111,148.584
C06991=1199.544,143.506,-53.200,-178.267,6.110,148.584
C06992=1199.549,143.257,-53.179,-178.270,6.108,148.585
C06993=1199.553,143.008,-53.159,-178.273,6.107,148.585
C06994=1199.558,142.758,-53.138,-178.275,6.106,148.586
C06995=1199.563,142.510,-53.117,-178.278,6.104,148.586
C06996=1199.568,142.260,-53.096,-178.280,6.102,148.586
C06997=1199.572,142.011,-53.076,-178.283,6.102,148.587
C06998=1199.577,141.762,-53.056,-178.286,6.100,148.587
C06999=1199.582,141.513,-53.035,-178.288,6.098,148.588
C07000=1199.587,141.264,-53.014,-178.291,6.097,148.588
C07001=1199.592,141.015,-52.993,-178.294,6.096,148.589
C07002=1199.596,140.766,-52.973,-178.296,6.094,148.589
C07003=1199.601,140.517,-52.953,-178.298,6.093,148.589
C07004=1199.606,140.268,-52.932,-178.302,6.091,148.590
C07005=1199.610,140.019,-52.911,-178.304,6.090,148.590
C07006=1199.615,139.770,-52.890,-178.306,6.089,148.591
C07007=1199.620,139.521,-52.870,-178.310,6.087,148.591
C07008=1199.625,139.271,-52.850,-178.312,6.085,148.592
C07009=1199.630,139.022,-52.829,-178.314,6.085,148.592
C07010=1199.634,138.773,-52.809,-178.318,6.083,148.593
C07011=1199.639,138.524,-52.788,-178.320,6.082,148.593
C07012=1199.644,138.275,-52.768,-178.322,6.080,148.594
C07013=1199.648,138.026,-52.747,-178.325,6.079,148.594
C07014=1199.653,137.777,-52.727,-178.328,6.078,148.595
C07015=1199.658,137.527,-52.707,-178.330,6.076,148.595
C07016=1199.663,137.278,-52.686,-178.333,6.074,148.595
C07017=1199.667,137.029,-52.666,-178.336,6.074,148.596
C07018=1199.671,136.780,-52.645,-178.338,6.072,148.596
C07019=1199.677,136.531,-52.624,-178.340,6.071,148.597
C07020=1199.681,136.281,-52.605,-178.344,6.070,148.597
C07021=1199.686,136.032,-52.584,-178.346,6.068,148.598
C07022=1199.691,135.783,-52.563,-178.348,6.067,148.598
C07023=1199.696,135.535,-52.543,-178.352,6.066,148.599
C07024=1199.701,135.285,-52.524,-178.354,6.064,148.599
C07025=1199.705,135.036,-52.503,-178.356,6.063,148.600
C07026=1199.710,134.787,-52.482,-178.359,6.061,148.600
C07027=1199.715,134.538,-52.462,-178.362,6.060,148.601
C07028=1199.720,134.288,-52.442,-178.364,6.059,148.601
C07029=1199.724,134.039,-52.422,-178.367,6.057,148.601
C07030=1199.728,133.790,-52.402,-178.370,6.056,148.602
C07031=1199.734,133.541,-52.381,-178.372,6.054,148.602
C07032=1199.738,133.273,-52.360,-178.375,6.053,148.603
C07033=1199.744,133.004,-52.338,-178.378,6.052,148.603
C07034=1199.749,132.736,-52.316,-178.381,6.051,148.604
C07035=1199.754,132.467,-52.294,-178.383,6.049,148.604
C07036=1199.759,132.218,-52.274,-178.386,6.047,148.605
C07037=1199.764,131.968,-52.254,-178.389,6.047,148.605
C07038=1199.768,131.719,-52.234,-178.391,6.045,148.606
C07039=1199.774,131.470,-52.214,-178.394,6.044,148.607
C07040=1199.779,131.221,-52.194,-178.397,6.042,148.607
C07041=1199.783,130.972,-52.173,-178.399,6.041,148.607
C07042=1199.788,130.722,-52.154,-178.402,6.040,148.608
C07043=1199.792,130.474,-52.133,-178.405,6.038,148.608
C07044=1199.797,130.224,-52.114,-178.407,6.037,148.609
C07045=1199.802,129.976,-52.094,-178.410,6.036,148.609
C07046=1199.807,129.726,-52.074,-178.412,6.035,148.610
C07047=1199.811,129.477,-52.054,-178.415,6.033,148.610
C07048=1199.817,129.227,-52.033,-178.418,6.032,148.611
C07049=1199.821,128.978,-52.013,-178.420,6.031,148.611
C07050=1199.826,128.730,-51.994,-178.423,6.029,148.612
C07051=1199.831,128.481,-51.973,-178.425,6.028,148.612
C07052=1199.836,128.231,-51.954,-178.428,6.027,148.613
C07053=1199.840,127.982,-51.933,-178.430,6.026,148.613
C07054=1199.845,127.732,-51.914,-178.433,6.024,148.614
C07055=1199.850,127.484,-51.894,-178.436,6.023,148.614
C07056=1199.855,127.235,-51.874,-178.439,6.022,148.615
C07057=1199.859,126.985,-51.854,-178.441,6.020,148.615
C07058=1199.864,126.736,-51.834,-178.443,6.019,148.615
C07059=1199.869,126.487,-51.815,-178.447,6.018,148.616
C07060=1199.874,126.238,-51.795,-178.449,6.017,148.616
C07061=1199.878,125.989,-51.775,-178.451,6.015,148.617
C07062=1199.883,125.739,-51.755,-178.454,6.014,148.617
C07063=1199.888,125.490,-51.736,-178.457,6.013,148.618
C07064=1199.893,125.241,-51.715,-178.460,6.011,148.618
C07065=1199.897,124.992,-51.696,-178.462,6.010,148.619
C07066=1199.902,124.742,-51.676,-178.465,6.009,148.619
C07067=1199.907,124.494,-51.656,-178.467,6.008,148.620
C07068=1199.912,124.244,-51.636,-178.470,6.006,148.620
C07069=1199.917,123.995,-51.617,-178.472,6.005,148.621
C07070=1199.921,123.746,-51.596,-178.475,6.004,148.621
C07071=1199.927,123.497,-51.577,-178.477,6.003,148.622
C07072=1199.931,123.248,-51.558,-178.481,6.001,148.622
C07073=1199.935,122.998,-51.538,-178.483,6.001,148.623
C07074=1199.940,122.750,-51.518,-178.485,5.999,148.623
C07075=1199.945,122.500,-51.499,-178.488,5.998,148.624
C07076=1199.950,122.251,-51.479,-178.491,5.996,148.624
C07077=1199.955,122.002,-51.460,-178.494,5.995,148.625
C07078=1199.960,121.752,-51.440,-178.496,5.994,148.625
C07079=1199.964,121.503,-51.420,-178.499,5.992,148.626
C07080=1199.970,121.255,-51.400,-178.501,5.992,148.626
C07081=1199.974,121.005,-51.381,-178.504,5.990,148.627
C07082=1199.978,120.756,-51.362,-178.507,5.989,148.627
C07083=1199.984,120.507,-51.342,-178.509,5.988,148.628
C07084=1199.989,120.257,-51.323,-178.512,5.987,148.628
C07085=1199.993,120.008,-51.302,-178.515,5.985,148.629
C07086=1199.998,119.760,-51.283,-178.517,5.984,148.629
C07087=1200.002,119.510,-51.264,-178.520,5.983,148.630
C07088=1200.007,119.261,-51.244,-178.522,5.982,148.630
C07089=1200.012,119.012,-51.225,-178.525,5.980,148.631
C07090=1200.017,118.762,-51.205,-178.527,5.980,148.631
C07091=1200.022,118.513,-51.186,-178.530,5.978,148.632
C07092=1200.026,118.264,-51.167,-178.533,5.977,148.632
C07093=1200.031,118.015,-51.147,-178.535,5.975,148.633
C07094=1200.037,117.766,-51.128,-178.538,5.975,148.633
C07095=1200.041,117.516,-51.109,-178.541,5.973,148.634
C07096=1200.046,117.267,-51.089,-178.543,5.972,148.634
C07097=1200.051,117.018,-51.070,-178.546,5.971,148.635
C07098=1200.055,116.768,-51.051,-178.548,5.970,148.635
C07099=1200.061,116.520,-51.031,-178.551,5.968,148.636
C07100=1200.065,116.270,-51.012,-178.553,5.967,148.636
C07101=1200.070,116.021,-50.993,-178.556,5.966,148.637
C07102=1200.075,115.772,-50.973,-178.559,5.965,148.637
C07103=1200.080,115.522,-50.954,-178.561,5.963,148.638
C07104=1200.084,115.274,-50.935,-178.564,5.963,148.638
C07105=1200.089,115.024,-50.915,-178.567,5.961,148.639
C07106=1200.094,114.775,-50.896,-178.569,5.960,148.639
C07107=1200.098,114.526,-50.877,-178.572,5.959,148.640
C07108=1200.104,114.277,-50.858,-178.574,5.958,148.640
C07109=1200.108,114.028,-50.838,-178.577,5.956,148.641
C07110=1200.114,113.779,-50.819,-178.579,5.955,148.641
C07111=1200.118,113.529,-50.800,-178.583,5.954,148.642
C07112=1200.123,113.279,-50.781,-178.585,5.953,148.642
C07113=1200.127,113.031,-50.762,-178.588,5.952,148.643
C07114=1200.132,112.781,-50.742,-178.590,5.951,148.643
C07115=1200.137,112.532,-50.723,-178.593,5.949,148.644
C07116=1200.141,112.283,-50.704,-178.595,5.948,148.644
C07117=1200.147,112.034,-50.685,-178.598,5.947,148.645
C07118=1200.152,111.784,-50.666,-178.601,5.946,148.645
C07119=1200.156,111.535,-50.647,-178.603,5.945,148.646
C07120=1200.161,111.286,-50.627,-178.606,5.944,148.646
C07121=1200.166,111.037,-50.609,-178.608,5.943,148.647
C07122=1200.171,110.787,-50.590,-178.611,5.941,148.647
C07123=1200.176,110.538,-50.570,-178.613,5.940,148.648
C07124=1200.180,110.289,-50.551,-178.617,5.939,148.648
C07125=1200.186,110.040,-50.532,-178.619,5.938,148.649
C07126=1200.190,109.790,-50.514,-178.622,5.937,148.649
C07127=1200.195,109.541,-50.494,-178.624,5.936,148.650
C07128=1200.200,109.293,-50.476,-178.627,5.935,148.651
C07129=1200.205,109.043,-50.457,-178.629,5.933,148.651
C07130=1200.209,108.794,-50.438,-178.632,5.932,148.651
C07131=1200.214,108.545,-50.418,-178.635,5.931,148.652
C07132=1200.219,108.295,-50.400,-178.637,5.930,148.652
C07133=1200.224,108.046,-50.381,-178.640,5.929,148.653
C07134=1200.229,107.797,-50.361,-178.642,5.928,148.653
C07135=1200.234,107.547,-50.343,-178.645,5.926,148.654
C07136=1200.239,107.279,-50.322,-178.647,5.925,148.654
C07137=1200.244,107.011,-50.303,-178.651,5.924,148.655
C07138=1200.249,106.742,-50.282,-178.653,5.923,148.656
C07139=1200.255,106.474,-50.262,-178.656,5.922,148.656
C07140=1200.259,106.224,-50.243,-178.659,5.920,148.657
C07141=1200.264,105.976,-50.224,-178.661,5.919,148.657
C07142=1200.269,105.726,-50.206,-178.664,5.919,148.658
C07143=1200.274,105.477,-50.186,-178.667,5.917,148.658
C07144=1200.279,105.228,-50.168,-178.669,5.916,148.659
C07145=1200.283,104.978,-50.149,-178.672,5.915,148.659
C07146=1200.288,104.729,-50.130,-178.675,5.914,148.660
C07147=1200.293,104.480,-50.112,-178.677,5.913,148.660
C07148=1200.298,104.230,-50.093,-178.680,5.912,148.661
C07149=1200.303,103.982,-50.074,-178.682,5.911,148.661
C07150=1200.308,103.732,-50.056,-178.685,5.909,148.662
C07151=1200.312,103.483,-50.036,-178.687,5.908,148.662
C07152=1200.317,103.234,-50.018,-178.691,5.907,148.663
C07153=1200.322,102.984,-49.999,-178.693,5.906,148.663
C07154=1200.327,102.735,-49.981,-178.695,5.906,148.664
C07155=1200.332,102.486,-49.962,-178.698,5.904,148.665
C07156=1200.337,102.236,-49.943,-178.701,5.903,148.665
C07157=1200.341,101.988,-49.924,-178.703,5.901,148.666
C07158=1200.346,101.738,-49.906,-178.706,5.901,148.666
C07159=1200.351,101.488,-49.887,-178.708,5.900,148.667
C07160=1200.356,101.240,-49.869,-178.711,5.899,148.667
C07161=1200.361,100.990,-49.851,-178.713,5.898,148.668
C07162=1200.365,100.741,-49.831,-178.717,5.896,148.668
C07163=1200.370,100.492,-49.813,-178.719,5.895,148.669
C07164=1200.375,100.243,-49.795,-178.721,5.895,148.669
C07165=1200.381,99.994,-49.776,-178.724,5.893,148.670
C07166=1200.385,99.744,-49.758,-178.727,5.892,148.670
C07167=1200.390,99.495,-49.740,-178.729,5.891,148.671
C07168=1200.395,99.246,-49.720,-178.732,5.890,148.672
C07169=1200.399,98.996,-49.702,-178.734,5.889,148.672
C07170=1200.404,98.747,-49.684,-178.737,5.888,148.673
C07171=1200.409,98.498,-49.665,-178.739,5.887,148.673
C07172=1200.414,98.248,-49.646,-178.743,5.885,148.674
C07173=1200.419,97.999,-49.628,-178.745,5.885,148.674
C07174=1200.424,97.750,-49.610,-178.747,5.884,148.675
C07175=1200.428,97.501,-49.592,-178.751,5.883,148.675
C07176=1200.433,97.251,-49.573,-178.753,5.882,148.676
C07177=1200.438,97.002,-49.555,-178.755,5.881,148.676
C07178=1200.443,96.753,-49.537,-178.758,5.879,148.677
C07179=1200.448,96.504,-49.518,-178.761,5.879,148.677
C07180=1200.452,96.254,-49.500,-178.763,5.877,148.678
C07181=1200.458,96.005,-49.481,-178.766,5.876,148.679
C07182=1200.463,95.755,-49.463,-178.768,5.875,148.679
C07183=1200.468,95.506,-49.445,-178.771,5.874,148.680
C07184=1200.472,95.258,-49.427,-178.773,5.873,148.680
C07185=1200.477,95.008,-49.408,-178.776,5.873,148.681
C07186=1200.482,94.759,-49.390,-178.779,5.871,148.681
C07187=1200.487,94.509,-49.372,-178.781,5.870,148.682
C07188=1200.492,94.260,-49.354,-178.784,5.870,148.682
C07189=1200.496,94.010,-49.335,-178.787,5.868,148.683
C07190=1200.501,93.761,-49.317,-178.789,5.867,148.683
C07191=1200.506,93.512,-49.299,-178.792,5.866,148.684
C07192=1200.511,93.263,-49.281,-178.795,5.865,148.684
C07193=1200.516,93.014,-49.263,-178.797,5.864,148.685
C07194=1200.521,92.764,-49.244,-178.800,5.863,148.686
C07195=1200.526,92.515,-49.226,-178.802,5.862,148.686
C07196=1200.531,92.265,-49.208,-178.805,5.861,148.687
C07197=1200.536,92.016,-49.190,-178.807,5.859,148.687
C07198=1200.540,91.767,-49.172,-178.810,5.859,148.688
C07199=1200.545,91.518,-49.154,-178.813,5.858,148.688
C07200=1200.550,91.268,-49.135,-178.815,5.857,148.689
C07201=1200.555,91.019,-49.117,-178.818,5.856,148.689
C07202=1200.559,90.770,-49.100,-178.820,5.855,148.690
C07203=1200.564,90.521,-49.082,-178.823,5.854,148.690
C07204=1200.569,90.271,-49.064,-178.825,5.853,148.691
C07205=1200.574,90.022,-49.046,-178.828,5.852,148.692
C07206=1200.579,89.773,-49.028,-178.831,5.850,148.692
C07207=1200.583,89.523,-49.009,-178.833,5.850,148.693
C07208=1200.588,89.274,-48.991,-178.836,5.849,148.693
C07209=1200.593,89.025,-48.973,-178.839,5.848,148.694
C07210=1200.598,88.776,-48.955,-178.841,5.847,148.694
C07211=1200.603,88.526,-48.937,-178.843,5.846,148.695
C07212=1200.608,88.277,-48.919,-178.847,5.845,148.695
C07213=1200.613,88.028,-48.901,-178.849,5.844,148.696
C07214=1200.618,87.778,-48.884,-178.851,5.843,148.696
C07215=1200.623,87.529,-48.866,-178.855,5.842,148.697
C07216=1200.627,87.279,-48.848,-178.857,5.841,148.698
C07217=1200.632,87.030,-48.830,-178.859,5.840,148.698
C07218=1200.637,86.781,-48.812,-178.862,5.839,148.699
C07219=1200.642,86.532,-48.794,-178.865,5.838,148.699
C07220=1200.647,86.283,-48.776,-178.867,5.837,148.700
C07221=1200.652,86.033,-48.759,-178.869,5.837,148.700
C07222=1200.657,85.784,-48.741,-178.873,5.835,148.701
C07223=1200.662,85.534,-48.723,-178.875,5.834,148.701
C07224=1200.667,85.285,-48.705,-178.877,5.834,148.702
C07225=1200.672,85.036,-48.687,-178.880,5.832,148.702
C07226=1200.677,84.786,-48.669,-178.883,5.831,148.703
C07227=1200.682,84.537,-48.651,-178.885,5.831,148.704
C07228=1200.686,84.288,-48.634,-178.888,5.829,148.704
C07229=1200.691,84.039,-48.616,-178.891,5.829,148.705
C07230=1200.696,83.789,-48.599,-178.893,5.828,148.705
C07231=1200.701,83.540,-48.581,-178.895,5.827,148.706
C07232=1200.706,83.290,-48.562,-178.898,5.825,148.706
C07233=1200.710,83.041,-48.544,-178.901,5.825,148.707
C07234=1200.716,82.791,-48.527,-178.903,5.824,148.708
C07235=1200.721,82.542,-48.509,-178.906,5.822,148.708
C07236=1200.725,82.293,-48.492,-178.909,5.822,148.709
C07237=1200.730,82.043,-48.475,-178.911,5.821,148.709
C07238=1200.735,81.794,-48.457,-178.914,5.820,148.710
C07239=1200.740,81.545,-48.439,-178.917,5.819,148.710
C07240=1200.746,81.277,-48.420,-178.919,5.818,148.711
C07241=1200.751,81.009,-48.401,-178.922,5.817,148.712
C07242=1200.756,80.740,-48.382,-178.925,5.816,148.712
C07243=1200.761,80.472,-48.363,-178.928,5.815,148.713
C07244=1200.766,80.222,-48.346,-178.930,5.814,148.713
C07245=1200.771,79.973,-48.328,-178.933,5.813,148.714
C07246=1200.776,79.724,-48.310,-178.935,5.813,148.715
C07247=1200.781,79.474,-48.293,-178.938,5.811,148.715
C07248=1200.785,79.225,-48.276,-178.941,5.810,148.716
C07249=1200.790,78.975,-48.258,-178.943,5.810,148.716
C07250=1200.795,78.726,-48.240,-178.946,5.808,148.717
C07251=1200.800,78.476,-48.223,-178.949,5.808,148.717
C07252=1200.805,78.228,-48.206,-178.951,5.807,148.718
C07253=1200.810,77.979,-48.188,-178.953,5.806,148.718
C07254=1200.815,77.729,-48.171,-178.957,5.805,148.719
C07255=1200.820,77.480,-48.153,-178.959,5.804,148.720
C07256=1200.825,77.230,-48.136,-178.961,5.803,148.720
C07257=1200.830,76.981,-48.118,-178.963,5.802,148.721
C07258=1200.835,76.731,-48.101,-178.967,5.801,148.721
C07259=1200.839,76.483,-48.083,-178.969,5.800,148.722
C07260=1200.844,76.233,-48.066,-178.971,5.799,148.722
C07261=1200.849,75.983,-48.049,-178.974,5.799,148.723
C07262=1200.854,75.734,-48.032,-178.977,5.798,148.724
C07263=1200.859,75.484,-48.014,-178.979,5.797,148.724
C07264=1200.864,75.236,-47.997,-178.982,5.796,148.725
C07265=1200.869,74.986,-47.980,-178.984,5.795,148.725
C07266=1200.874,74.737,-47.962,-178.987,5.794,148.726
C07267=1200.879,74.487,-47.945,-178.990,5.793,148.727
C07268=1200.883,74.238,-47.928,-178.992,5.792,148.727
C07269=1200.888,73.989,-47.910,-178.995,5.792,148.728
C07270=1200.894,73.739,-47.893,-178.998,5.790,148.728
C07271=1200.898,73.490,-47.875,-179.000,5.789,148.729
C07272=1200.903,73.240,-47.858,-179.003,5.789,148.729
C07273=1200.908,72.992,-47.842,-179.005,5.788,148.730
C07274=1200.913,72.742,-47.824,-179.008,5.787,148.730
C07275=1200.918,72.493,-47.807,-179.011,5.786,148.731
C07276=1200.923,72.243,-47.790,-179.013,5.785,148.732
C07277=1200.928,71.994,-47.772,-179.015,5.785,148.732
C07278=1200.932,71.744,-47.755,-179.018,5.784,148.733
C07279=1200.938,71.495,-47.738,-179.021,5.782,148.733
C07280=1200.942,71.246,-47.722,-179.023,5.782,148.734
C07281=1200.947,70.997,-47.704,-179.026,5.781,148.735
C07282=1200.952,70.747,-47.687,-179.028,5.780,148.735
C07283=1200.957,70.497,-47.670,-179.031,5.779,148.736
C07284=1200.962,70.248,-47.653,-179.034,5.778,148.736
C07285=1200.967,69.999,-47.636,-179.036,5.777,148.737
C07286=1200.972,69.750,-47.618,-179.039,5.777,148.737
C07287=1200.977,69.500,-47.602,-179.041,5.776,148.738
C07288=1200.982,69.250,-47.584,-179.044,5.775,148.739
C07289=1200.986,69.001,-47.567,-179.047,5.774,148.739
C07290=1200.992,68.752,-47.550,-179.049,5.773,148.740
C07291=1200.996,68.503,-47.533,-179.052,5.773,148.740
C07292=1201.002,68.253,-47.516,-179.055,5.771,148.741
C07293=1201.006,68.004,-47.499,-179.057,5.770,148.741
C07294=1201.012,67.755,-47.483,-179.060,5.770,148.742
C07295=1201.016,67.506,-47.465,-179.062,5.769,148.743
C07296=1201.021,67.256,-47.448,-179.064,5.768,148.743
C07297=1201.026,67.006,-47.431,-179.068,5.767,148.744
C07298=1201.030,66.757,-47.415,-179.070,5.766,148.744
